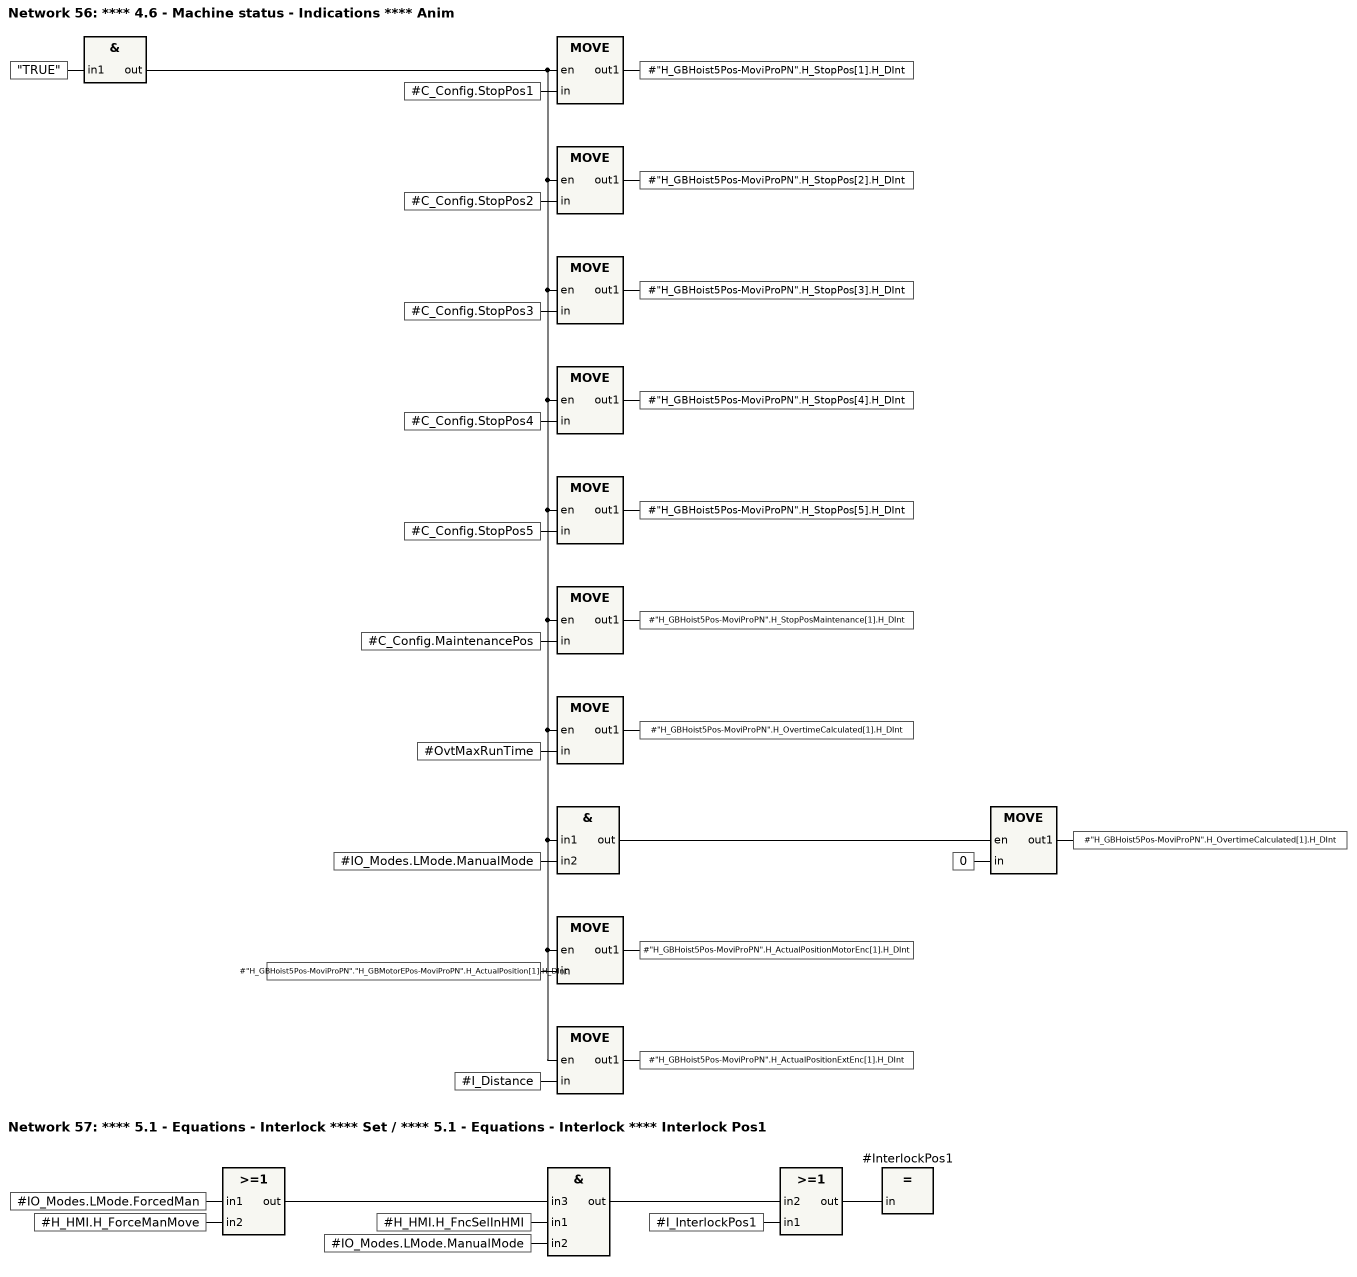
   IF "TRUE" THEN
       #"H_GBHoist5Pos-MoviProPN".H_StopPos[1].H_DInt := #C_Config.StopPos1;
       #"H_GBHoist5Pos-MoviProPN".H_StopPos[2].H_DInt := #C_Config.StopPos2;
       #"H_GBHoist5Pos-MoviProPN".H_StopPos[3].H_DInt := #C_Config.StopPos3;
       #"H_GBHoist5Pos-MoviProPN".H_StopPos[4].H_DInt := #C_Config.StopPos4;
       #"H_GBHoist5Pos-MoviProPN".H_StopPos[5].H_DInt := #C_Config.StopPos5;
       #"H_GBHoist5Pos-MoviProPN".H_StopPosMaintenance[1].H_DInt := #C_Config.MaintenancePos;
       #"H_GBHoist5Pos-MoviProPN".H_OvertimeCalculated[1].H_DInt := #OvtMaxRunTime;
   END_IF;
   IF "TRUE" AND #IO_Modes.LMode.ManualMode THEN
       #"H_GBHoist5Pos-MoviProPN".H_OvertimeCalculated[1].H_DInt := 0;
   END_IF;
   IF "TRUE" THEN
       #"H_GBHoist5Pos-MoviProPN".H_ActualPositionMotorEnc[1].H_DInt := #"H_GBHoist5Pos-MoviProPN"."H_GBMotorEPos-MoviProPN".H_ActualPosition[1].H_DInt;
       #"H_GBHoist5Pos-MoviProPN".H_ActualPositionExtEnc[1].H_DInt := #I_Distance;
   END_IF;
END_REGION

REGION Network 57: **** 5.1 - Equations - Interlock **** Set / **** 5.1 - Equations - Interlock **** Interlock Pos1
   // Interlock
   #InterlockPos1 := ((#IO_Modes.LMode.ForcedMan OR #H_HMI.H_ForceManMove) AND #H_HMI.H_FncSelInHMI AND #IO_Modes.LMode.ManualMode) OR #I_InterlockPos1;
END_REGION

REGION Network 58: **** 5.1 - Equations - Interlock **** Set / **** 5.1 - Equations - Interlock **** Interlock Pos2
   // Interlock
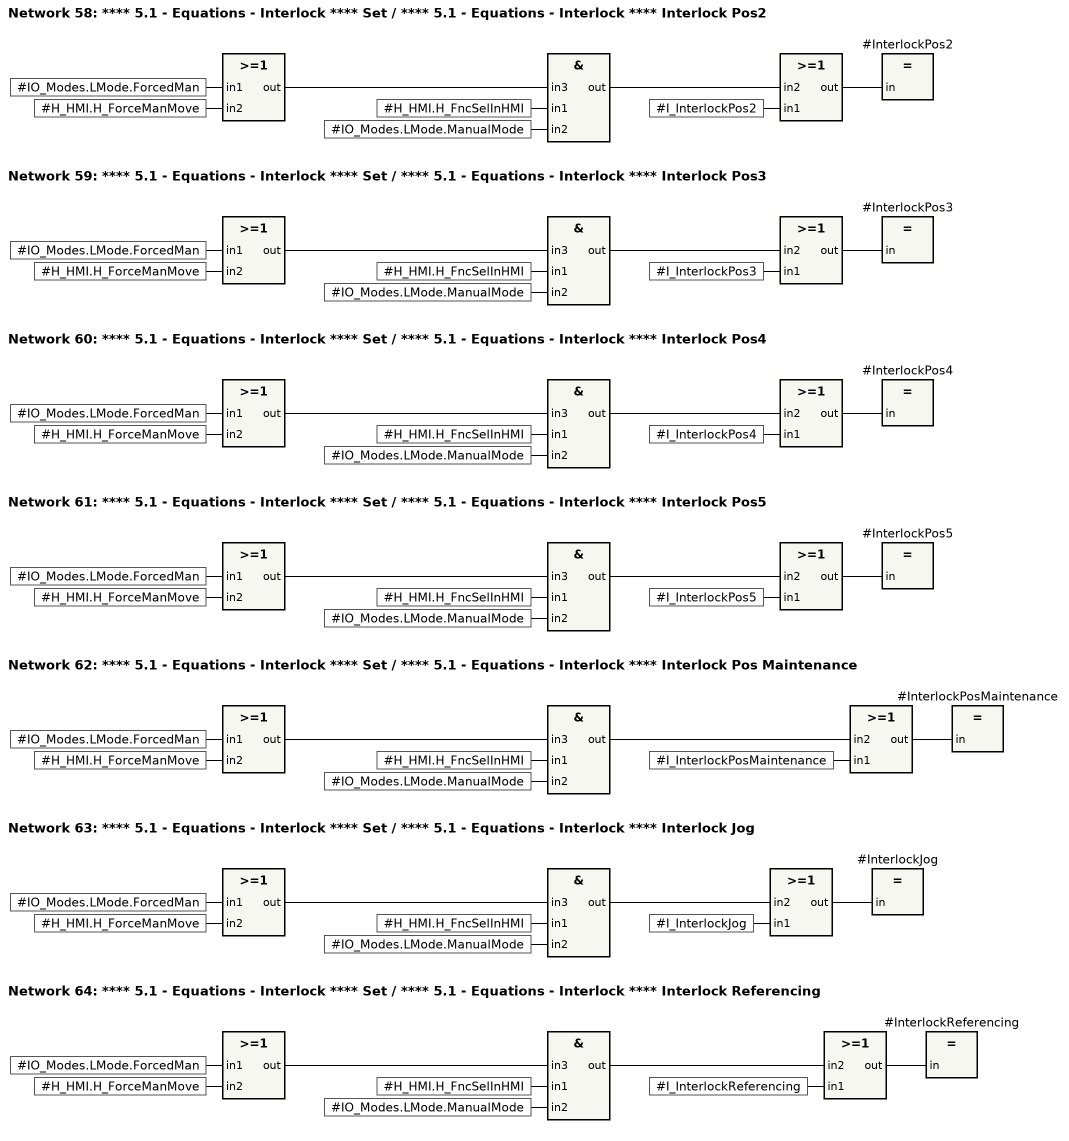
   #InterlockPos2 := ((#IO_Modes.LMode.ForcedMan OR #H_HMI.H_ForceManMove) AND #H_HMI.H_FncSelInHMI AND #IO_Modes.LMode.ManualMode) OR #I_InterlockPos2;
END_REGION

REGION Network 59: **** 5.1 - Equations - Interlock **** Set / **** 5.1 - Equations - Interlock **** Interlock Pos3
   // Interlock
   #InterlockPos3 := ((#IO_Modes.LMode.ForcedMan OR #H_HMI.H_ForceManMove) AND #H_HMI.H_FncSelInHMI AND #IO_Modes.LMode.ManualMode) OR #I_InterlockPos3;
END_REGION

REGION Network 60: **** 5.1 - Equations - Interlock **** Set / **** 5.1 - Equations - Interlock **** Interlock Pos4
   // Interlock
   #InterlockPos4 := ((#IO_Modes.LMode.ForcedMan OR #H_HMI.H_ForceManMove) AND #H_HMI.H_FncSelInHMI AND #IO_Modes.LMode.ManualMode) OR #I_InterlockPos4;
END_REGION

REGION Network 61: **** 5.1 - Equations - Interlock **** Set / **** 5.1 - Equations - Interlock **** Interlock Pos5
   // Interlock
   #InterlockPos5 := ((#IO_Modes.LMode.ForcedMan OR #H_HMI.H_ForceManMove) AND #H_HMI.H_FncSelInHMI AND #IO_Modes.LMode.ManualMode) OR #I_InterlockPos5;
END_REGION

REGION Network 62: **** 5.1 - Equations - Interlock **** Set / **** 5.1 - Equations - Interlock **** Interlock Pos Maintenance
   // Interlock
   #InterlockPosMaintenance := ((#IO_Modes.LMode.ForcedMan OR #H_HMI.H_ForceManMove) AND #H_HMI.H_FncSelInHMI AND #IO_Modes.LMode.ManualMode) OR #I_InterlockPosMaintenance;
END_REGION

REGION Network 63: **** 5.1 - Equations - Interlock **** Set / **** 5.1 - Equations - Interlock **** Interlock Jog
   // Interlock
   #InterlockJog := ((#IO_Modes.LMode.ForcedMan OR #H_HMI.H_ForceManMove) AND #H_HMI.H_FncSelInHMI AND #IO_Modes.LMode.ManualMode) OR #I_InterlockJog;
END_REGION

REGION Network 64: **** 5.1 - Equations - Interlock **** Set / **** 5.1 - Equations - Interlock **** Interlock Referencing
   // Interlock
   #InterlockReferencing := ((#IO_Modes.LMode.ForcedMan OR #H_HMI.H_ForceManMove) AND #H_HMI.H_FncSelInHMI AND #IO_Modes.LMode.ManualMode) OR #I_InterlockReferencing;
END_REGION

REGION Network 65: **** 5.2 - Equations - Equations **** Epos Cmd
   // Drive is steered by EPos commands
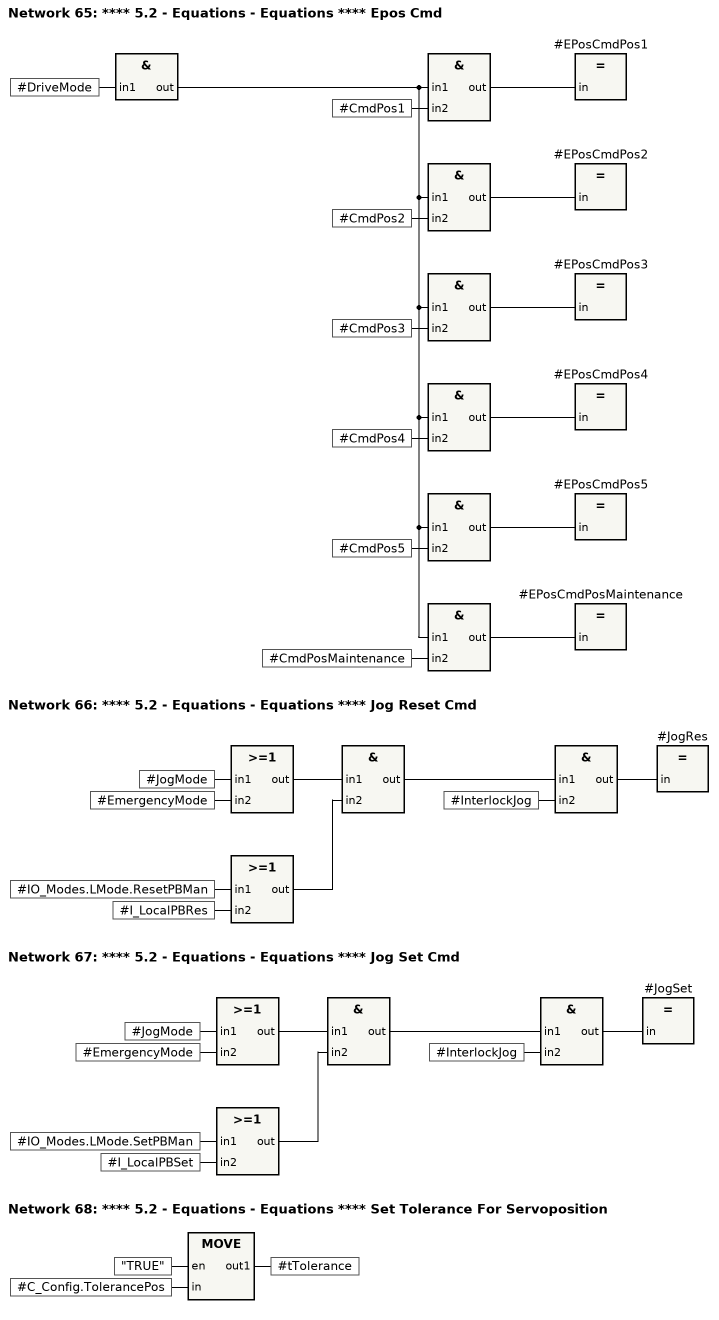
   #EPosCmdPos1 := #DriveMode AND #CmdPos1;
   #EPosCmdPos2 := #DriveMode AND #CmdPos2;
   #EPosCmdPos3 := #DriveMode AND #CmdPos3;
   #EPosCmdPos4 := #DriveMode AND #CmdPos4;
   #EPosCmdPos5 := #DriveMode AND #CmdPos5;
   #EPosCmdPosMaintenance := #DriveMode AND #CmdPosMaintenance;
END_REGION

REGION Network 66: **** 5.2 - Equations - Equations **** Jog Reset Cmd
   // Drive is steered by Jog commands in reset direction
   #JogRes := (#JogMode OR #EmergencyMode) AND (#IO_Modes.LMode.ResetPBMan OR #I_LocalPBRes) AND #InterlockJog;
END_REGION

REGION Network 67: **** 5.2 - Equations - Equations **** Jog Set Cmd
   // Drive is steered by Jog commands in set direction
   #JogSet := (#JogMode OR #EmergencyMode) AND (#IO_Modes.LMode.SetPBMan OR #I_LocalPBSet) AND #InterlockJog;
END_REGION

REGION Network 68: **** 5.2 - Equations - Equations **** Set Tolerance For Servoposition
   // Set Tolerance For ServoPosition
   IF "TRUE" THEN #tTolerance := #C_Config.TolerancePos; END_IF;
END_REGION

REGION Network 69: **** 5.2 - Equations - Equations **** Calculate Tolerance Index Pos 1
   // Calculate Tolerance Index Pos 1
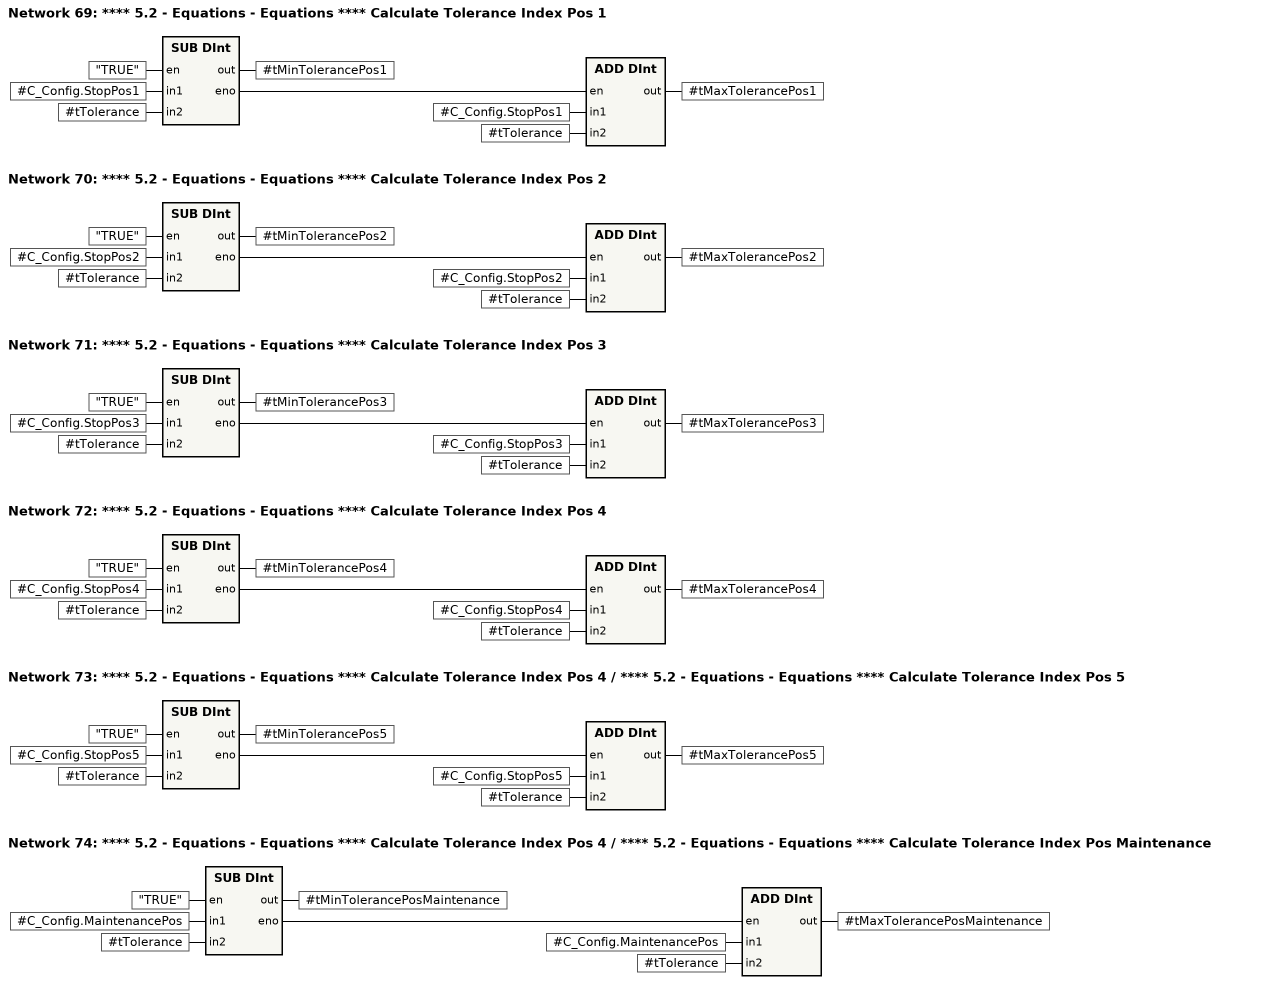
   // ENO of a box is taken as its EN; it also drops when the box reports an error
   IF "TRUE" THEN
       #tMinTolerancePos1 := #C_Config.StopPos1 - #tTolerance;
       #tMaxTolerancePos1 := #C_Config.StopPos1 + #tTolerance;
   END_IF;
END_REGION

REGION Network 70: **** 5.2 - Equations - Equations **** Calculate Tolerance Index Pos 2
   // Calculate Tolerance Index Pos 2
   // ENO of a box is taken as its EN; it also drops when the box reports an error
   IF "TRUE" THEN
       #tMinTolerancePos2 := #C_Config.StopPos2 - #tTolerance;
       #tMaxTolerancePos2 := #C_Config.StopPos2 + #tTolerance;
   END_IF;
END_REGION

REGION Network 71: **** 5.2 - Equations - Equations **** Calculate Tolerance Index Pos 3
   // Calculate Tolerance Index Pos 3
   // ENO of a box is taken as its EN; it also drops when the box reports an error
   IF "TRUE" THEN
       #tMinTolerancePos3 := #C_Config.StopPos3 - #tTolerance;
       #tMaxTolerancePos3 := #C_Config.StopPos3 + #tTolerance;
   END_IF;
END_REGION

REGION Network 72: **** 5.2 - Equations - Equations **** Calculate Tolerance Index Pos 4
   // Calculate Tolerance Index Pos 4
   // ENO of a box is taken as its EN; it also drops when the box reports an error
   IF "TRUE" THEN
       #tMinTolerancePos4 := #C_Config.StopPos4 - #tTolerance;
       #tMaxTolerancePos4 := #C_Config.StopPos4 + #tTolerance;
   END_IF;
END_REGION

REGION Network 73: **** 5.2 - Equations - Equations **** Calculate Tolerance Index Pos 4 / **** 5.2 - Equations - Equations **** Calculate Tolerance Index Pos 5
   // Calculate Tolerance Index Pos 4 / Calculate Tolerance Index Pos 5
   // ENO of a box is taken as its EN; it also drops when the box reports an error
   IF "TRUE" THEN
       #tMinTolerancePos5 := #C_Config.StopPos5 - #tTolerance;
       #tMaxTolerancePos5 := #C_Config.StopPos5 + #tTolerance;
   END_IF;
END_REGION

REGION Network 74: **** 5.2 - Equations - Equations **** Calculate Tolerance Index Pos 4 / **** 5.2 - Equations - Equations **** Calculate Tolerance Index Pos Maintenance
   // Calculate Tolerance Index Pos 4 / Calculate Tolerance Index Pos Maintenance
   // ENO of a box is taken as its EN; it also drops when the box reports an error
   IF "TRUE" THEN
       #tMinTolerancePosMaintenance := #C_Config.MaintenancePos - #tTolerance;
       #tMaxTolerancePosMaintenance := #C_Config.MaintenancePos + #tTolerance;
   END_IF;
END_REGION

REGION Network 75: **** 5.2 - Equations - Equations **** Alarm Condition Keep Position 1
   // Alarm Condition Keep Position
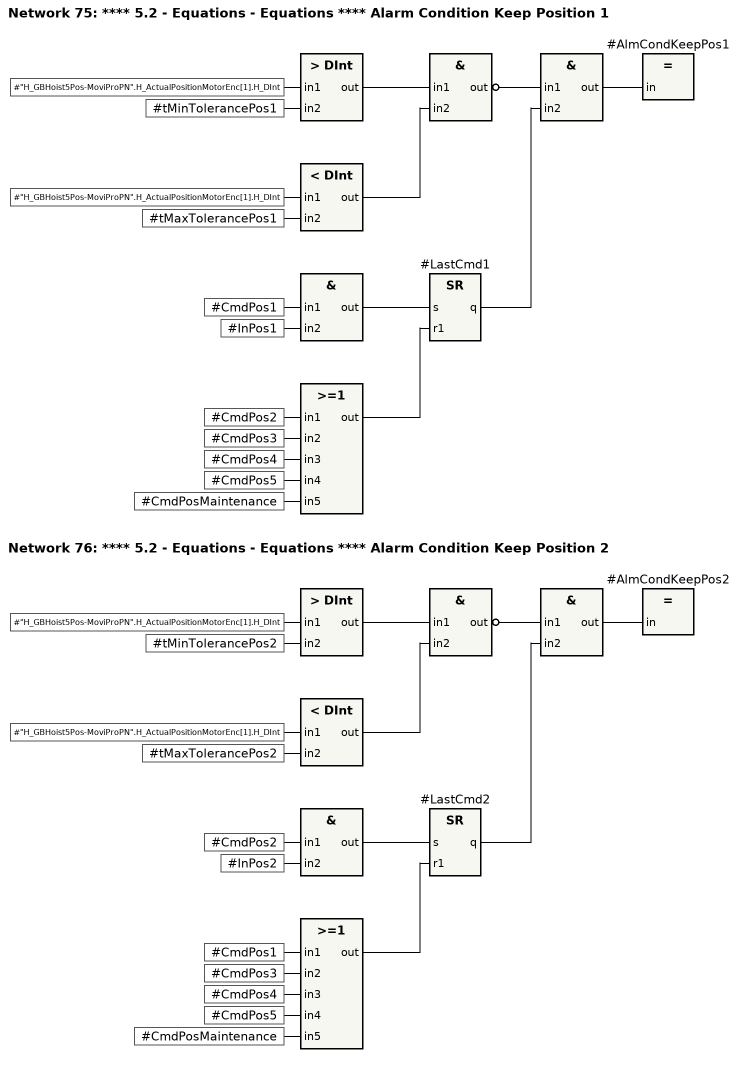
   IF #CmdPos1 AND #InPos1 THEN
       #LastCmd1 := TRUE;   // SR flip-flop
   END_IF;
   IF #CmdPos2 OR #CmdPos3 OR #CmdPos4 OR #CmdPos5 OR #CmdPosMaintenance THEN #LastCmd1 := FALSE; END_IF;
   #AlmCondKeepPos1 := NOT ((#"H_GBHoist5Pos-MoviProPN".H_ActualPositionMotorEnc[1].H_DInt > #tMinTolerancePos1) AND (#"H_GBHoist5Pos-MoviProPN".H_ActualPositionMotorEnc[1].H_DInt < #tMaxTolerancePos1)) AND #LastCmd1;
END_REGION

REGION Network 76: **** 5.2 - Equations - Equations **** Alarm Condition Keep Position 2
   // Alarm Condition Keep Position
   IF #CmdPos2 AND #InPos2 THEN
       #LastCmd2 := TRUE;   // SR flip-flop
   END_IF;
   IF #CmdPos1 OR #CmdPos3 OR #CmdPos4 OR #CmdPos5 OR #CmdPosMaintenance THEN #LastCmd2 := FALSE; END_IF;
   #AlmCondKeepPos2 := NOT ((#"H_GBHoist5Pos-MoviProPN".H_ActualPositionMotorEnc[1].H_DInt > #tMinTolerancePos2) AND (#"H_GBHoist5Pos-MoviProPN".H_ActualPositionMotorEnc[1].H_DInt < #tMaxTolerancePos2)) AND #LastCmd2;
END_REGION

REGION Network 77: **** 5.2 - Equations - Equations **** Alarm Condition Keep Position 3
   // Alarm Condition Keep Position
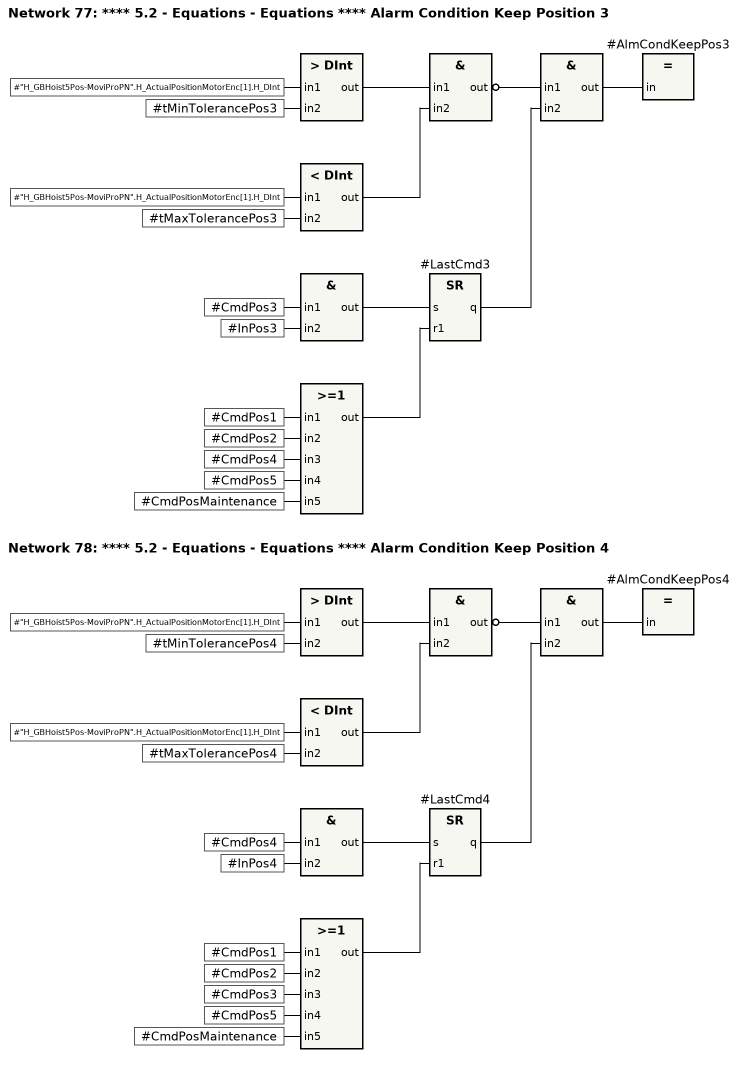
   IF #CmdPos3 AND #InPos3 THEN
       #LastCmd3 := TRUE;   // SR flip-flop
   END_IF;
   IF #CmdPos1 OR #CmdPos2 OR #CmdPos4 OR #CmdPos5 OR #CmdPosMaintenance THEN #LastCmd3 := FALSE; END_IF;
   #AlmCondKeepPos3 := NOT ((#"H_GBHoist5Pos-MoviProPN".H_ActualPositionMotorEnc[1].H_DInt > #tMinTolerancePos3) AND (#"H_GBHoist5Pos-MoviProPN".H_ActualPositionMotorEnc[1].H_DInt < #tMaxTolerancePos3)) AND #LastCmd3;
END_REGION

REGION Network 78: **** 5.2 - Equations - Equations **** Alarm Condition Keep Position 4
   // Alarm Condition Keep Position
   IF #CmdPos4 AND #InPos4 THEN
       #LastCmd4 := TRUE;   // SR flip-flop
   END_IF;
   IF #CmdPos1 OR #CmdPos2 OR #CmdPos3 OR #CmdPos5 OR #CmdPosMaintenance THEN #LastCmd4 := FALSE; END_IF;
   #AlmCondKeepPos4 := NOT ((#"H_GBHoist5Pos-MoviProPN".H_ActualPositionMotorEnc[1].H_DInt > #tMinTolerancePos4) AND (#"H_GBHoist5Pos-MoviProPN".H_ActualPositionMotorEnc[1].H_DInt < #tMaxTolerancePos4)) AND #LastCmd4;
END_REGION

REGION Network 79: **** 5.2 - Equations - Equations **** Alarm Condition Keep Position 4 / **** 5.2 - Equations - Equations **** Alarm Condition Keep Position 5
   // Alarm Condition Keep Position
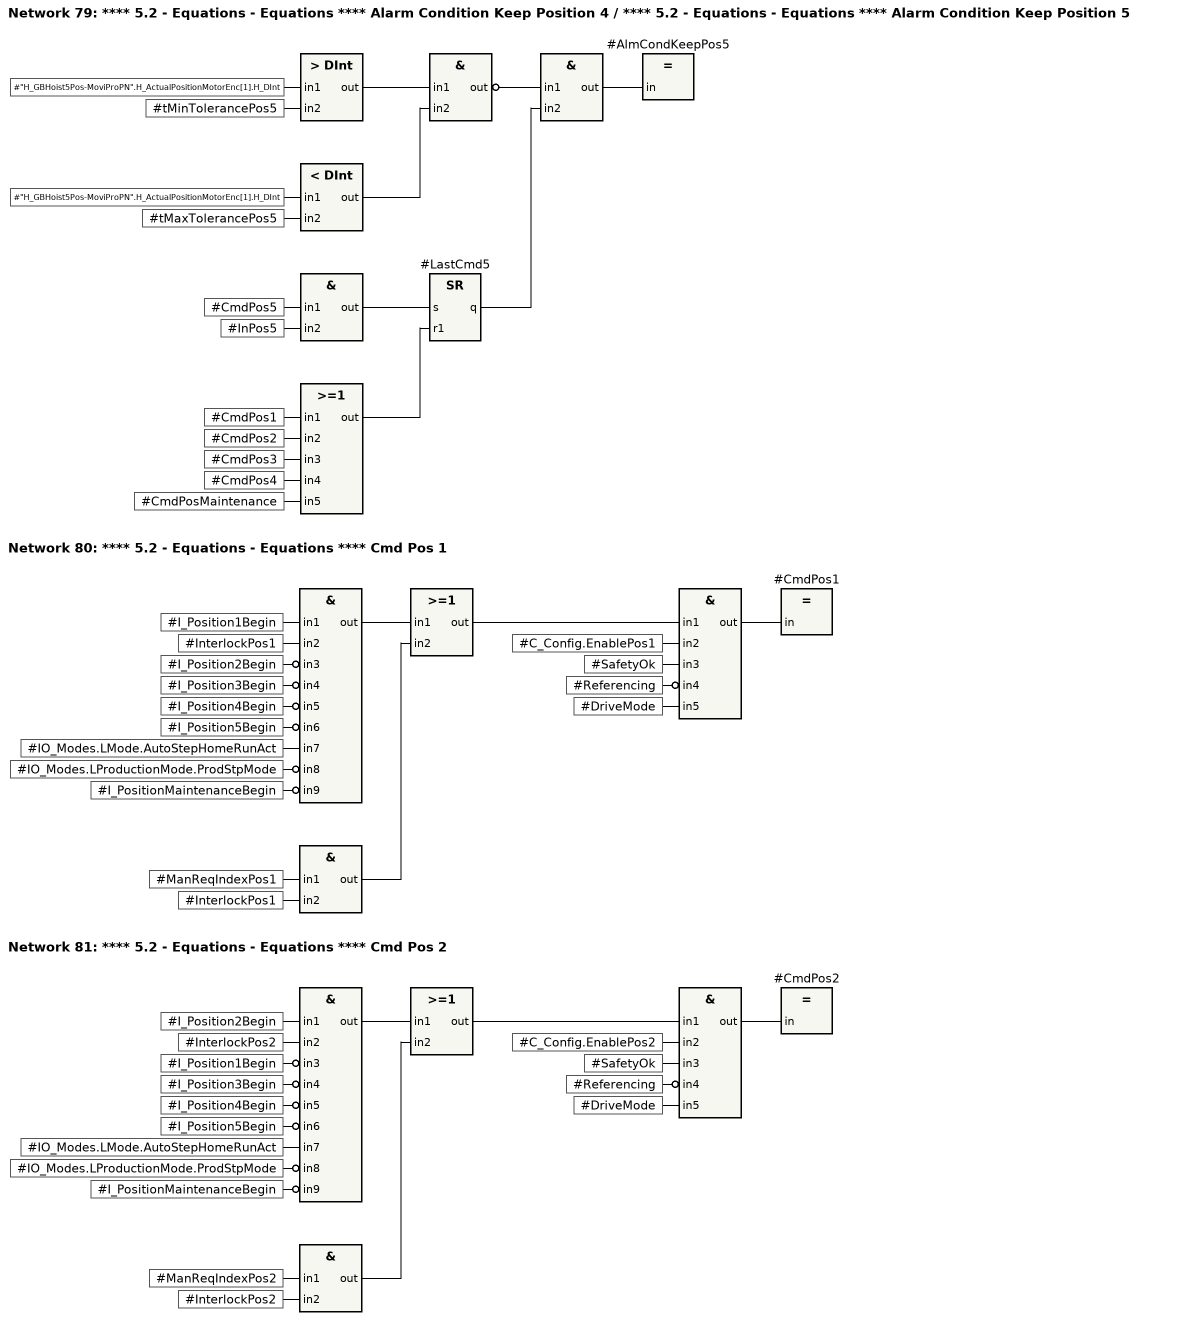
   IF #CmdPos5 AND #InPos5 THEN
       #LastCmd5 := TRUE;   // SR flip-flop
   END_IF;
   IF #CmdPos1 OR #CmdPos2 OR #CmdPos3 OR #CmdPos4 OR #CmdPosMaintenance THEN #LastCmd5 := FALSE; END_IF;
   #AlmCondKeepPos5 := NOT ((#"H_GBHoist5Pos-MoviProPN".H_ActualPositionMotorEnc[1].H_DInt > #tMinTolerancePos5) AND (#"H_GBHoist5Pos-MoviProPN".H_ActualPositionMotorEnc[1].H_DInt < #tMaxTolerancePos5)) AND #LastCmd5;
END_REGION

REGION Network 80: **** 5.2 - Equations - Equations **** Cmd Pos 1
   // Cmd Pos 1
   #CmdPos1 := ((#I_Position1Begin AND #InterlockPos1 AND NOT #I_Position2Begin AND NOT #I_Position3Begin AND NOT #I_Position4Begin AND NOT #I_Position5Begin AND #IO_Modes.LMode.AutoStepHomeRunAct AND NOT #IO_Modes.LProductionMode.ProdStpMode AND NOT #I_PositionMaintenanceBegin) OR (#ManReqIndexPos1 AND #InterlockPos1)) AND #C_Config.EnablePos1 AND #SafetyOk AND NOT #Referencing AND #DriveMode;
END_REGION

REGION Network 81: **** 5.2 - Equations - Equations **** Cmd Pos 2
   // Cmd Pos 2
   #CmdPos2 := ((#I_Position2Begin AND #InterlockPos2 AND NOT #I_Position1Begin AND NOT #I_Position3Begin AND NOT #I_Position4Begin AND NOT #I_Position5Begin AND #IO_Modes.LMode.AutoStepHomeRunAct AND NOT #IO_Modes.LProductionMode.ProdStpMode AND NOT #I_PositionMaintenanceBegin) OR (#ManReqIndexPos2 AND #InterlockPos2)) AND #C_Config.EnablePos2 AND #SafetyOk AND NOT #Referencing AND #DriveMode;
END_REGION

REGION Network 82: **** 5.2 - Equations - Equations **** Cmd Pos 3
   // Cmd Pos 3
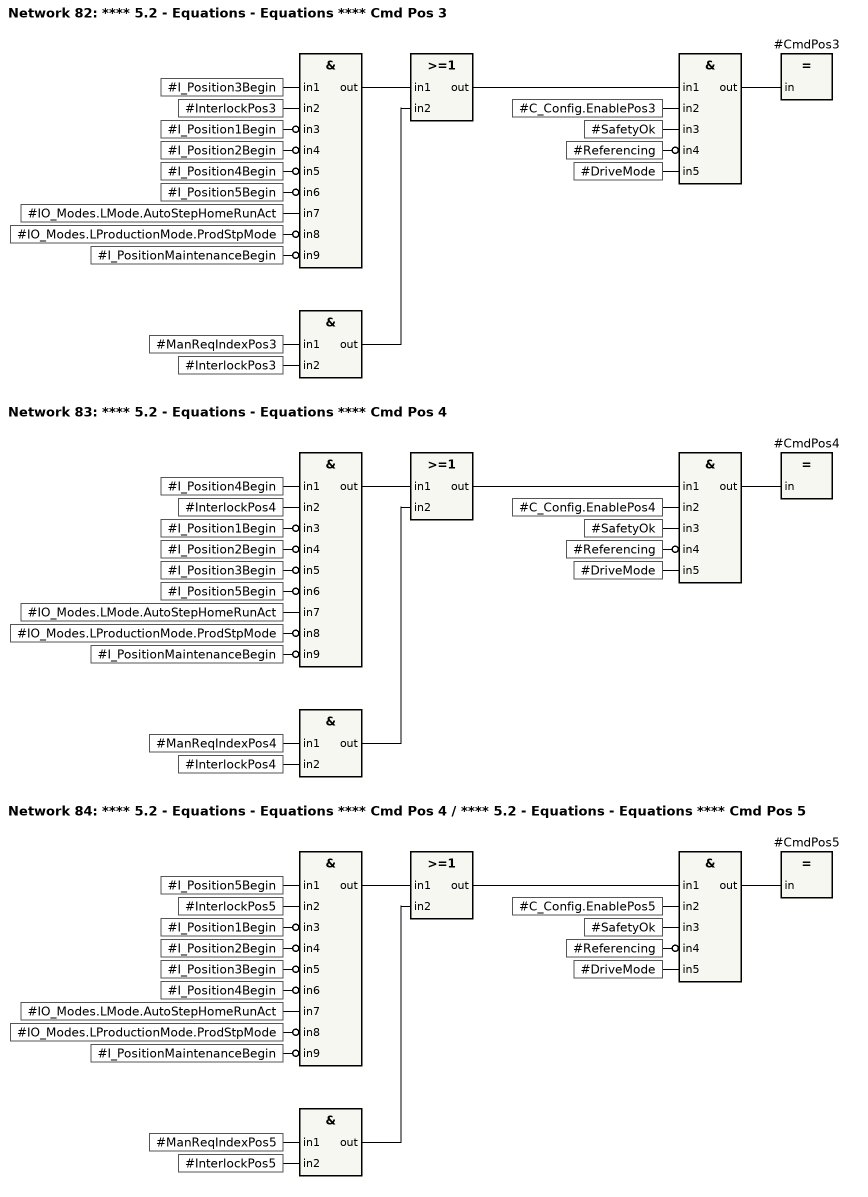
   #CmdPos3 := ((#I_Position3Begin AND #InterlockPos3 AND NOT #I_Position1Begin AND NOT #I_Position2Begin AND NOT #I_Position4Begin AND NOT #I_Position5Begin AND #IO_Modes.LMode.AutoStepHomeRunAct AND NOT #IO_Modes.LProductionMode.ProdStpMode AND NOT #I_PositionMaintenanceBegin) OR (#ManReqIndexPos3 AND #InterlockPos3)) AND #C_Config.EnablePos3 AND #SafetyOk AND NOT #Referencing AND #DriveMode;
END_REGION

REGION Network 83: **** 5.2 - Equations - Equations **** Cmd Pos 4
   // Cmd Pos 4
   #CmdPos4 := ((#I_Position4Begin AND #InterlockPos4 AND NOT #I_Position1Begin AND NOT #I_Position2Begin AND NOT #I_Position3Begin AND NOT #I_Position5Begin AND #IO_Modes.LMode.AutoStepHomeRunAct AND NOT #IO_Modes.LProductionMode.ProdStpMode AND NOT #I_PositionMaintenanceBegin) OR (#ManReqIndexPos4 AND #InterlockPos4)) AND #C_Config.EnablePos4 AND #SafetyOk AND NOT #Referencing AND #DriveMode;
END_REGION

REGION Network 84: **** 5.2 - Equations - Equations **** Cmd Pos 4 / **** 5.2 - Equations - Equations **** Cmd Pos 5
   // Cmd Pos 4
   #CmdPos5 := ((#I_Position5Begin AND #InterlockPos5 AND NOT #I_Position1Begin AND NOT #I_Position2Begin AND NOT #I_Position3Begin AND NOT #I_Position4Begin AND #IO_Modes.LMode.AutoStepHomeRunAct AND NOT #IO_Modes.LProductionMode.ProdStpMode AND NOT #I_PositionMaintenanceBegin) OR (#ManReqIndexPos5 AND #InterlockPos5)) AND #C_Config.EnablePos5 AND #SafetyOk AND NOT #Referencing AND #DriveMode;
END_REGION

REGION Network 85: **** 5.2 - Equations - Equations **** Cmd Pos 4 / **** 5.2 - Equations - Equations **** Cmd Pos Maintenance
   // Cmd Pos 4 / Cmd Pos Maintenance
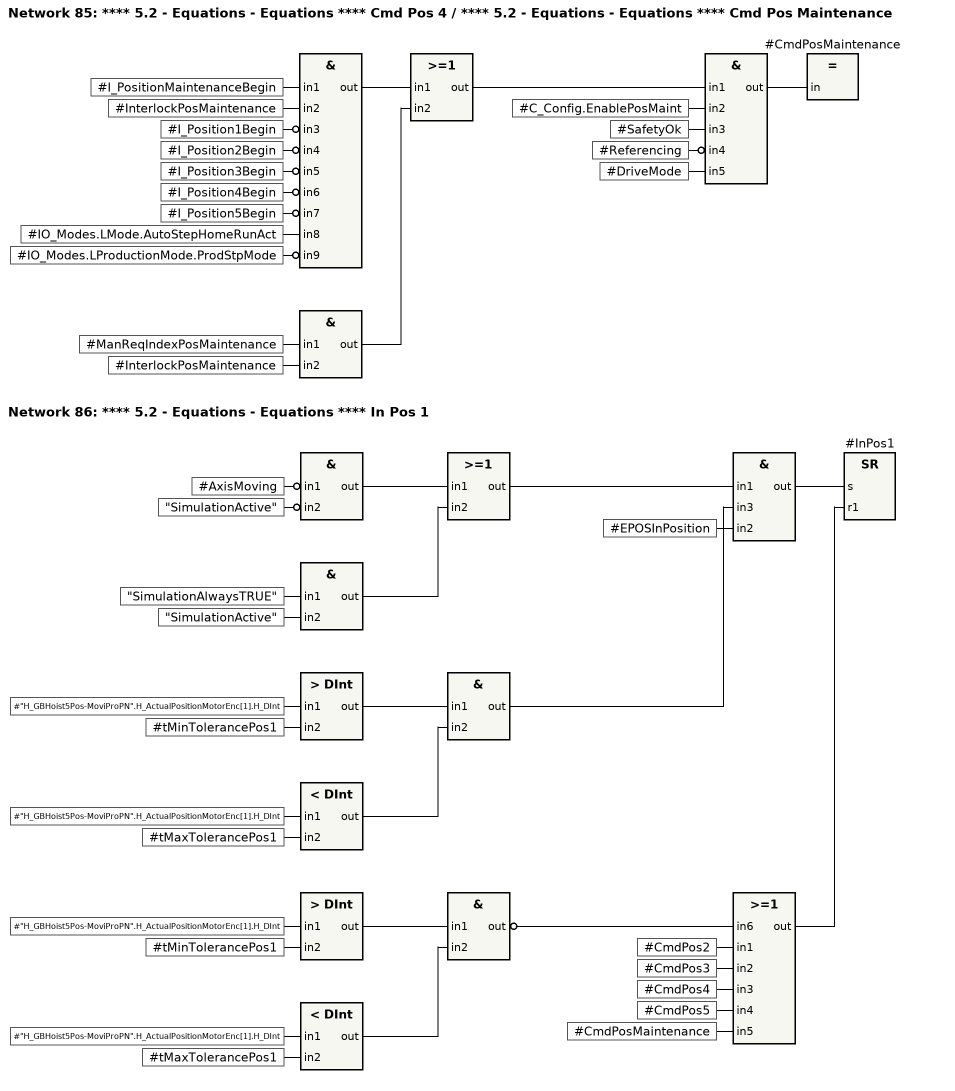
   #CmdPosMaintenance := ((#I_PositionMaintenanceBegin AND #InterlockPosMaintenance AND NOT #I_Position1Begin AND NOT #I_Position2Begin AND NOT #I_Position3Begin AND NOT #I_Position4Begin AND NOT #I_Position5Begin AND #IO_Modes.LMode.AutoStepHomeRunAct AND NOT #IO_Modes.LProductionMode.ProdStpMode) OR (#ManReqIndexPosMaintenance AND #InterlockPosMaintenance)) AND #C_Config.EnablePosMaint AND #SafetyOk AND NOT #Referencing AND #DriveMode;
END_REGION

REGION Network 86: **** 5.2 - Equations - Equations **** In Pos 1
   // In Pos 1
   IF ((NOT #AxisMoving AND NOT "SimulationActive") OR ("SimulationAlwaysTRUE" AND "SimulationActive")) AND (#"H_GBHoist5Pos-MoviProPN".H_ActualPositionMotorEnc[1].H_DInt > #tMinTolerancePos1) AND (#"H_GBHoist5Pos-MoviProPN".H_ActualPositionMotorEnc[1].H_DInt < #tMaxTolerancePos1) AND #EPOSInPosition THEN
       #InPos1 := TRUE;   // SR flip-flop
   END_IF;
   IF NOT ((#"H_GBHoist5Pos-MoviProPN".H_ActualPositionMotorEnc[1].H_DInt > #tMinTolerancePos1) AND (#"H_GBHoist5Pos-MoviProPN".H_ActualPositionMotorEnc[1].H_DInt < #tMaxTolerancePos1)) OR #CmdPos2 OR #CmdPos3 OR #CmdPos4 OR #CmdPos5 OR #CmdPosMaintenance THEN
       #InPos1 := FALSE;
   END_IF;
END_REGION

REGION Network 87: **** 5.2 - Equations - Equations **** In Pos 2
   // In Pos 2
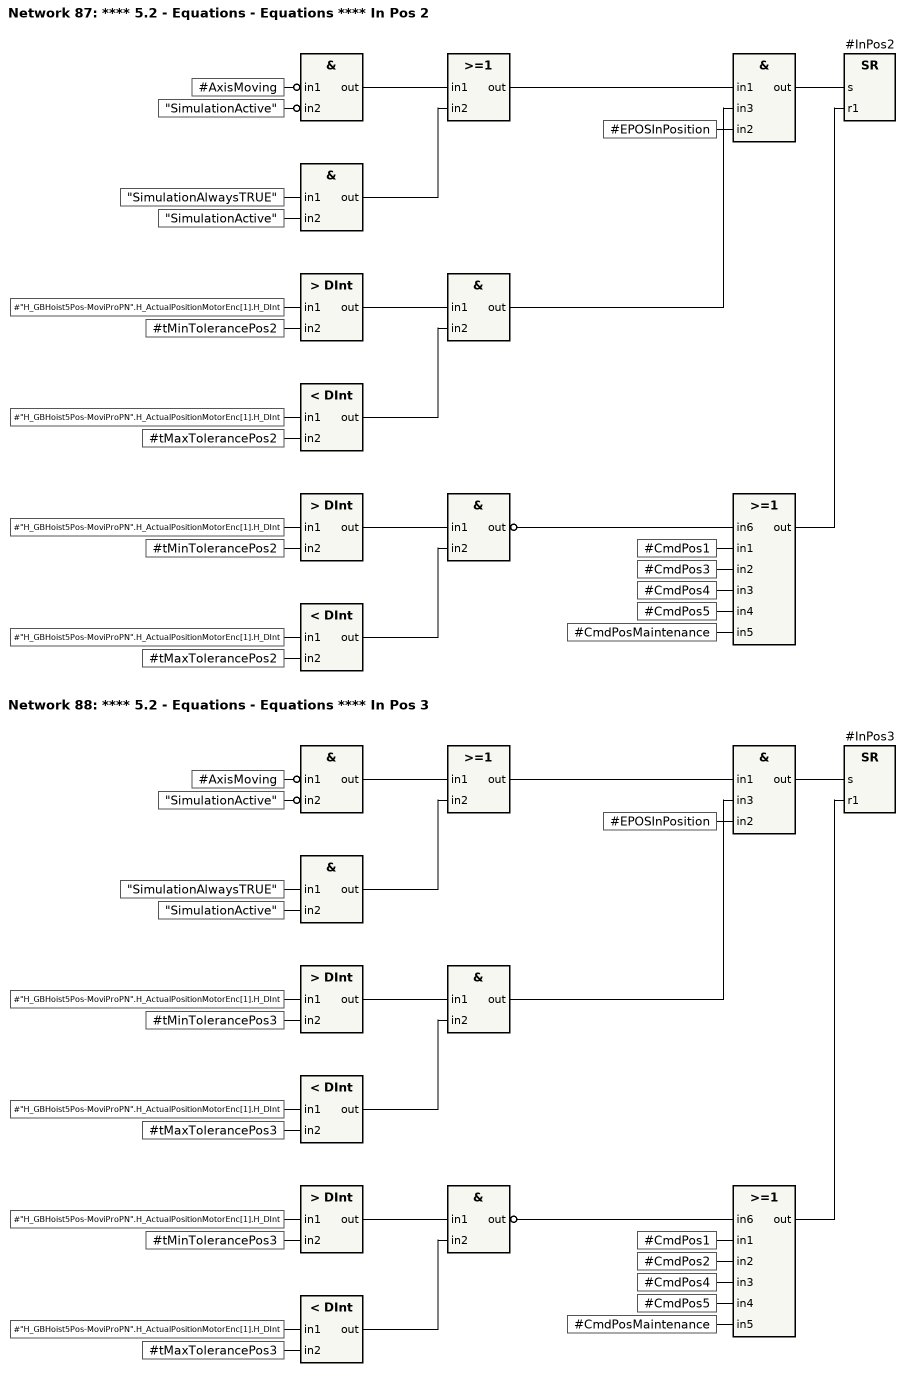
   IF ((NOT #AxisMoving AND NOT "SimulationActive") OR ("SimulationAlwaysTRUE" AND "SimulationActive")) AND (#"H_GBHoist5Pos-MoviProPN".H_ActualPositionMotorEnc[1].H_DInt > #tMinTolerancePos2) AND (#"H_GBHoist5Pos-MoviProPN".H_ActualPositionMotorEnc[1].H_DInt < #tMaxTolerancePos2) AND #EPOSInPosition THEN
       #InPos2 := TRUE;   // SR flip-flop
   END_IF;
   IF NOT ((#"H_GBHoist5Pos-MoviProPN".H_ActualPositionMotorEnc[1].H_DInt > #tMinTolerancePos2) AND (#"H_GBHoist5Pos-MoviProPN".H_ActualPositionMotorEnc[1].H_DInt < #tMaxTolerancePos2)) OR #CmdPos1 OR #CmdPos3 OR #CmdPos4 OR #CmdPos5 OR #CmdPosMaintenance THEN
       #InPos2 := FALSE;
   END_IF;
END_REGION

REGION Network 88: **** 5.2 - Equations - Equations **** In Pos 3
   // In Pos 3
   IF ((NOT #AxisMoving AND NOT "SimulationActive") OR ("SimulationAlwaysTRUE" AND "SimulationActive")) AND (#"H_GBHoist5Pos-MoviProPN".H_ActualPositionMotorEnc[1].H_DInt > #tMinTolerancePos3) AND (#"H_GBHoist5Pos-MoviProPN".H_ActualPositionMotorEnc[1].H_DInt < #tMaxTolerancePos3) AND #EPOSInPosition THEN
       #InPos3 := TRUE;   // SR flip-flop
   END_IF;
   IF NOT ((#"H_GBHoist5Pos-MoviProPN".H_ActualPositionMotorEnc[1].H_DInt > #tMinTolerancePos3) AND (#"H_GBHoist5Pos-MoviProPN".H_ActualPositionMotorEnc[1].H_DInt < #tMaxTolerancePos3)) OR #CmdPos1 OR #CmdPos2 OR #CmdPos4 OR #CmdPos5 OR #CmdPosMaintenance THEN
       #InPos3 := FALSE;
   END_IF;
END_REGION

REGION Network 89: **** 5.2 - Equations - Equations **** In Pos 4
   // In Pos 4
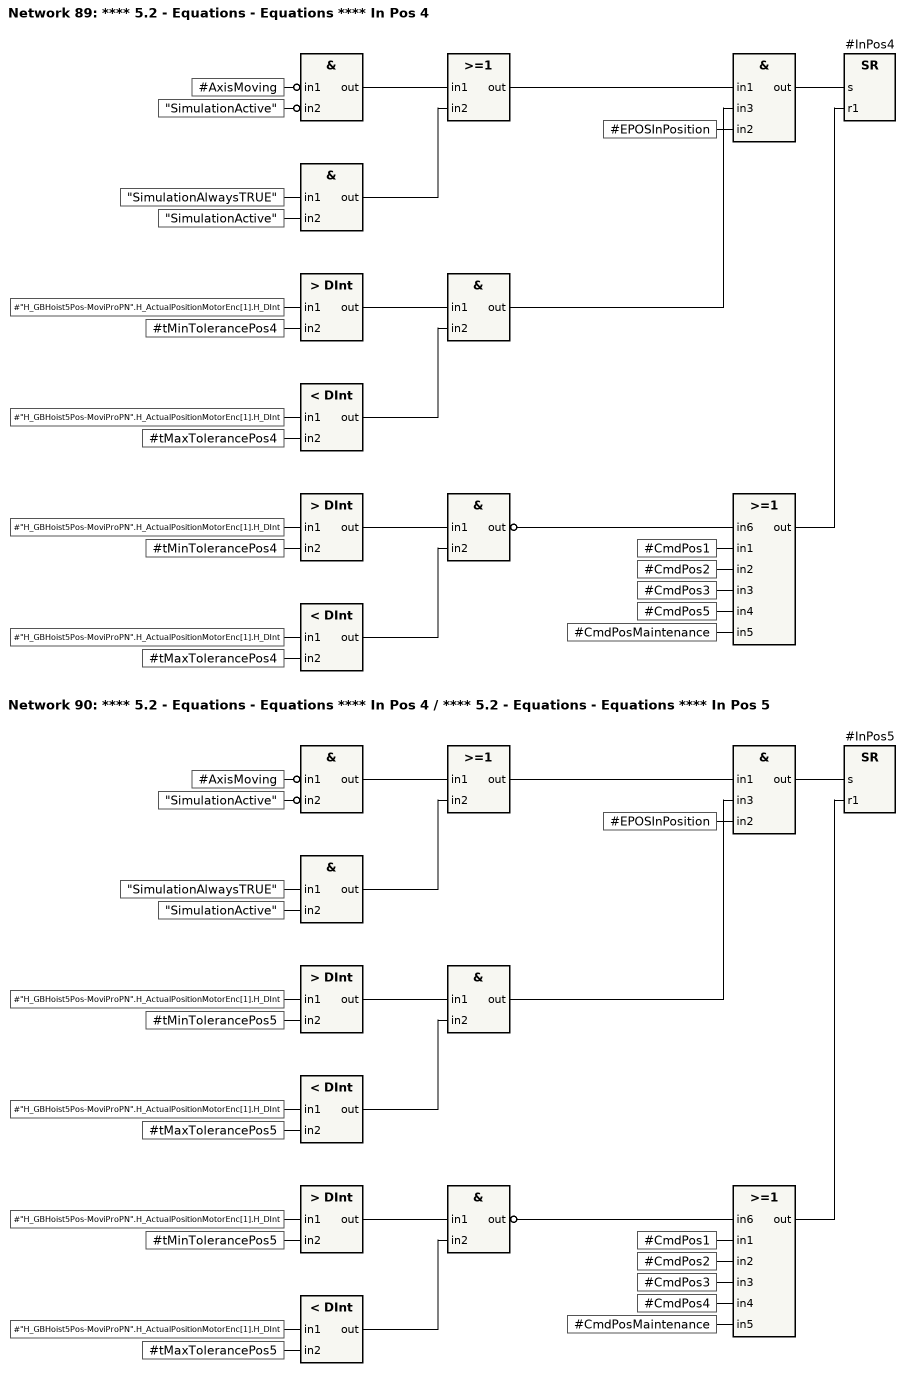
   IF ((NOT #AxisMoving AND NOT "SimulationActive") OR ("SimulationAlwaysTRUE" AND "SimulationActive")) AND (#"H_GBHoist5Pos-MoviProPN".H_ActualPositionMotorEnc[1].H_DInt > #tMinTolerancePos4) AND (#"H_GBHoist5Pos-MoviProPN".H_ActualPositionMotorEnc[1].H_DInt < #tMaxTolerancePos4) AND #EPOSInPosition THEN
       #InPos4 := TRUE;   // SR flip-flop
   END_IF;
   IF NOT ((#"H_GBHoist5Pos-MoviProPN".H_ActualPositionMotorEnc[1].H_DInt > #tMinTolerancePos4) AND (#"H_GBHoist5Pos-MoviProPN".H_ActualPositionMotorEnc[1].H_DInt < #tMaxTolerancePos4)) OR #CmdPos1 OR #CmdPos2 OR #CmdPos3 OR #CmdPos5 OR #CmdPosMaintenance THEN
       #InPos4 := FALSE;
   END_IF;
END_REGION

REGION Network 90: **** 5.2 - Equations - Equations **** In Pos 4 / **** 5.2 - Equations - Equations **** In Pos 5
   // In Pos 4 / In Pos 5
   IF ((NOT #AxisMoving AND NOT "SimulationActive") OR ("SimulationAlwaysTRUE" AND "SimulationActive")) AND (#"H_GBHoist5Pos-MoviProPN".H_ActualPositionMotorEnc[1].H_DInt > #tMinTolerancePos5) AND (#"H_GBHoist5Pos-MoviProPN".H_ActualPositionMotorEnc[1].H_DInt < #tMaxTolerancePos5) AND #EPOSInPosition THEN
       #InPos5 := TRUE;   // SR flip-flop
   END_IF;
   IF NOT ((#"H_GBHoist5Pos-MoviProPN".H_ActualPositionMotorEnc[1].H_DInt > #tMinTolerancePos5) AND (#"H_GBHoist5Pos-MoviProPN".H_ActualPositionMotorEnc[1].H_DInt < #tMaxTolerancePos5)) OR #CmdPos1 OR #CmdPos2 OR #CmdPos3 OR #CmdPos4 OR #CmdPosMaintenance THEN
       #InPos5 := FALSE;
   END_IF;
END_REGION

REGION Network 91: **** 5.2 - Equations - Equations **** In Pos 4 / **** 5.2 - Equations - Equations **** In Pos Maintenance
   // In Pos 4 / In Pos Maintenance
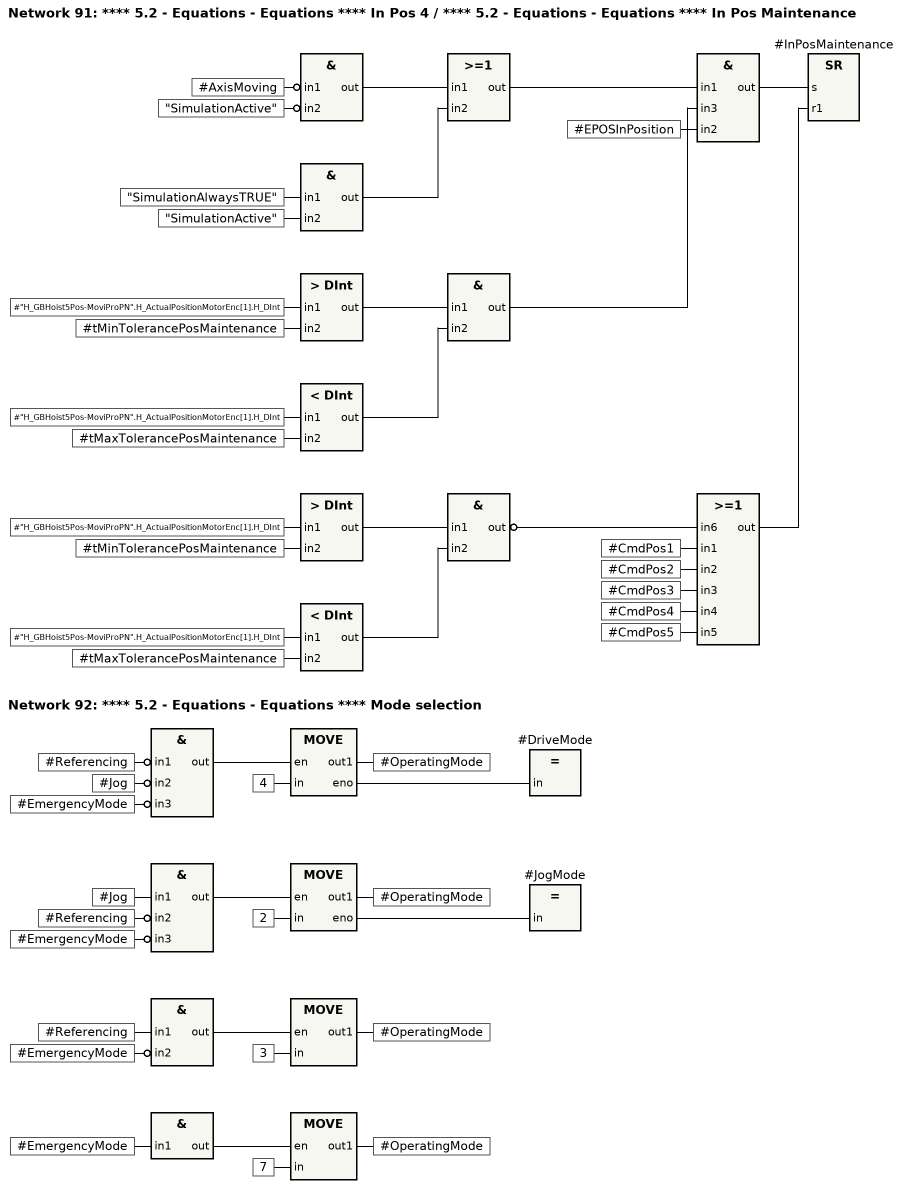
   IF ((NOT #AxisMoving AND NOT "SimulationActive") OR ("SimulationAlwaysTRUE" AND "SimulationActive")) AND (#"H_GBHoist5Pos-MoviProPN".H_ActualPositionMotorEnc[1].H_DInt > #tMinTolerancePosMaintenance) AND (#"H_GBHoist5Pos-MoviProPN".H_ActualPositionMotorEnc[1].H_DInt < #tMaxTolerancePosMaintenance) AND #EPOSInPosition THEN
       #InPosMaintenance := TRUE;   // SR flip-flop
   END_IF;
   IF NOT ((#"H_GBHoist5Pos-MoviProPN".H_ActualPositionMotorEnc[1].H_DInt > #tMinTolerancePosMaintenance) AND (#"H_GBHoist5Pos-MoviProPN".H_ActualPositionMotorEnc[1].H_DInt < #tMaxTolerancePosMaintenance)) OR #CmdPos1 OR #CmdPos2 OR #CmdPos3 OR #CmdPos4 OR #CmdPos5 THEN
       #InPosMaintenance := FALSE;
   END_IF;
END_REGION

REGION Network 92: **** 5.2 - Equations - Equations **** Mode selection
   #_w1 := NOT #Referencing AND NOT #Jog AND NOT #EmergencyMode;
   IF #_w1 THEN #OperatingMode := 4; END_IF;
   #DriveMode := #_w1;
   #_w2 := #Jog AND NOT #Referencing AND NOT #EmergencyMode;
   IF #_w2 THEN
       #OperatingMode := 2;   // Mode selection bits mode: 0=Default 1=Speed control 2=Jog mode 3=Referencing mode 4=Positioning mode 5=Positioning mode - touch probe 6=Speed synchronization 7=Emergency mode _
   END_IF;
   #JogMode := #_w2;
   IF #Referencing AND NOT #EmergencyMode THEN #OperatingMode := 3; END_IF;
   IF #EmergencyMode THEN #OperatingMode := 7; END_IF;
END_REGION

REGION Network 93: **** 5.2 - Equations - Equations **** Start command
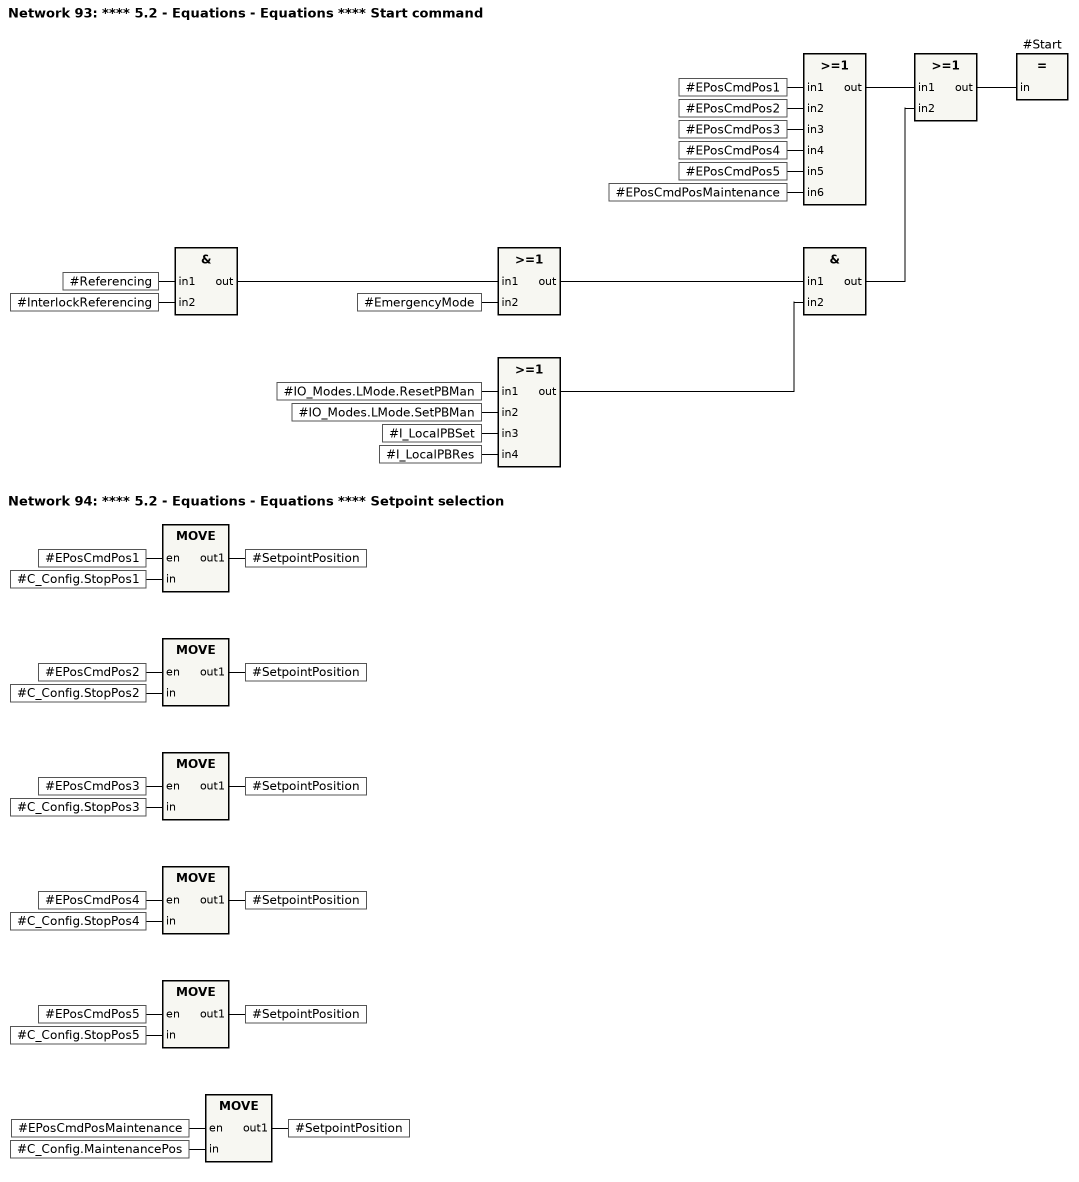
   #Start := #EPosCmdPos1 OR #EPosCmdPos2 OR #EPosCmdPos3 OR #EPosCmdPos4 OR #EPosCmdPos5 OR #EPosCmdPosMaintenance OR (((#Referencing AND #InterlockReferencing) OR #EmergencyMode) AND (#IO_Modes.LMode.ResetPBMan OR #IO_Modes.LMode.SetPBMan OR #I_LocalPBSet OR #I_LocalPBRes));
END_REGION

REGION Network 94: **** 5.2 - Equations - Equations **** Setpoint selection
   IF #EPosCmdPos1 THEN #SetpointPosition := #C_Config.StopPos1; END_IF;
   IF #EPosCmdPos2 THEN #SetpointPosition := #C_Config.StopPos2; END_IF;
   IF #EPosCmdPos3 THEN #SetpointPosition := #C_Config.StopPos3; END_IF;
   IF #EPosCmdPos4 THEN #SetpointPosition := #C_Config.StopPos4; END_IF;
   IF #EPosCmdPos5 THEN #SetpointPosition := #C_Config.StopPos5; END_IF;
   IF #EPosCmdPosMaintenance THEN #SetpointPosition := #C_Config.MaintenancePos; END_IF;
END_REGION

REGION Network 95: **** 7.3 - Submodule - Machine **** Motorloop
   // Motor loop
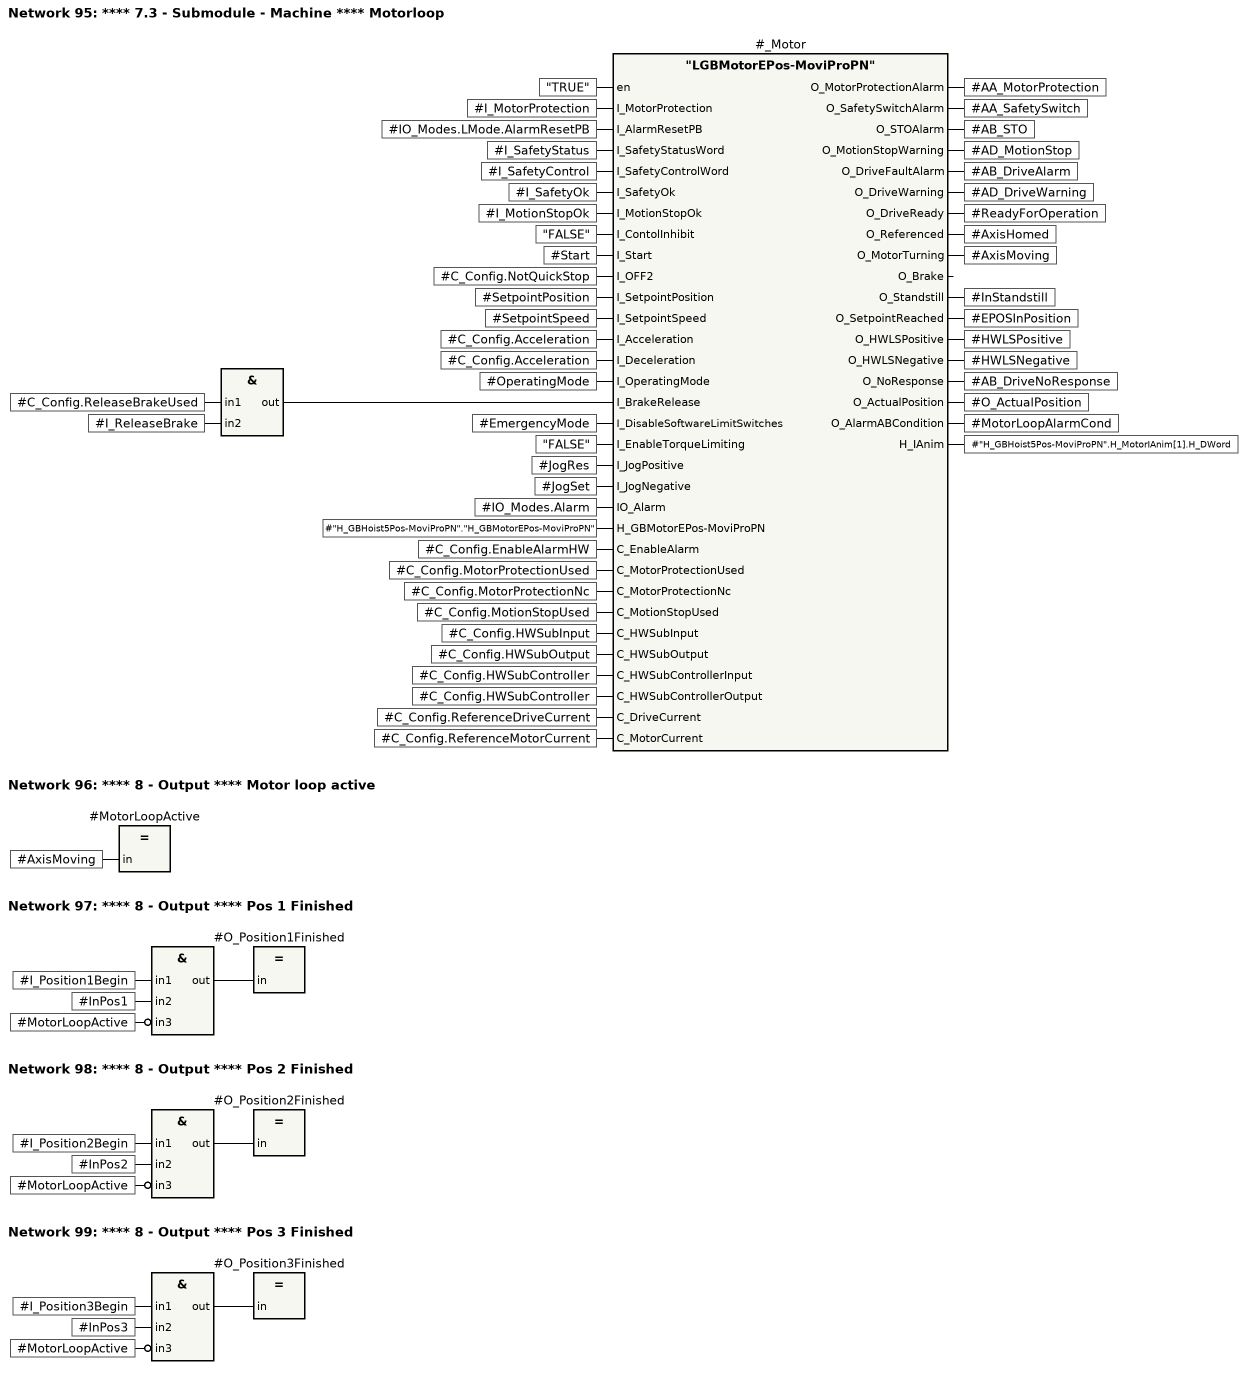
   IF "TRUE" THEN
       #_Motor(I_MotorProtection := #I_MotorProtection,   // "LGBMotorEPos-MoviProPN": Quick stop "I_OFF2" : ^ Speed (%) Stop signal at 5s l / 100% l______________/_ l \ \ l \ \ l \ \ l \ \ 0% l___________________\_____\___________________________> Time (s) l OFF2 OFF1 (regular start stop) 7s 10s ************************************************************************************ "I_SetpointSpeed" , "I_Acceleration", "I_Deceleration": Speed Target speed (user unit) ^ / l ____/____ l / \ l / \ l____/ \____ l--------------------------------------------------> t (s) Speed (user unit) ^ Acceleration l l _________ l l / \ l l/ \ l____/ \____ l--------------------------------------------------> t (s) Speed (user unit) ^ Deceleration l _________ l l / \ l l / \l l____/ \____ l--------------------------------------------------> t (s) ************************************************************************************ Mode selection bits "I_OperatingMode" : mode: 0=Default 1=Speed control 2=Jog mode 3=Referencing mode 4=Positioning mode 5=Positioning mode - touch probe 6=Speed synchronization 7=Emergency mode ************************************************************************************ Software limit switches "I_DisbaleSoftwareLimitSwitches" : The software limit switches are programmed before the hardware limit switches. This will give the drive the possiblility to decelarate accordingly as its knows the distance to these SW LS's from the encoder value. When the referencing is ok it should be impossible to reach the hardware limit switches. Only when there is a faulty referencing then the software limit switches can be behind the hardware limit switch. In that case it is possible to hit the hardware limit switch with full speed. Positive <-- Load --> negative HW LS SW LS _____ SW LS HW LS ____ ____ l_____l ____ ____ l____\ l____\ l_____l /____l /____l OOOOOOOOOOOOOOOOOOOOOOOOOOOOOOOOOOOO ll // \\ ll ll// \\ll ll ll ************************************************************************************ Input "I_EnableTorqueLimiting" : 110% ^ Torque (%) l Torque limited 100% l_______________________________/___________________ torque limit configured in the drive l _ Acceleration l l l l l / l l---- shutdown command l l l/ constant speed l l (error motor blocked) l l l_____/__ l l 0% l___l_________l________________l__l___________________________> Time (s) l l l l l l l / l l l / l_l -100% l __________ /________________________________________ torque limit configured in the drive l Deceleration -110% l ************************************************************************************ Communication handeling is done in the block with the "C_HWSub..." hardware identifiers. SEW Drive ______________ ll __ _ ll__ input telegram ll l__l l_l ll Ol ===============>> PLC ll ll__l ll_____________ll l__l l__l l_ll_l SEW Drive ______________ output telegram ll __ _ ll__ PLC ===============>> ll l__l l_l ll Ol ll ll__l ll_____________ll l__l l__l l_ll_l _
               I_AlarmResetPB := #IO_Modes.LMode.AlarmResetPB,
               I_SafetyStatusWord := #I_SafetyStatus,
               I_SafetyControlWord := #I_SafetyControl,
               I_SafetyOk := #I_SafetyOk,
               I_MotionStopOk := #I_MotionStopOk,
               I_ContolInhibit := "FALSE",
               I_Start := #Start,
               I_OFF2 := #C_Config.NotQuickStop,
               I_SetpointPosition := #SetpointPosition,
               I_SetpointSpeed := #SetpointSpeed,
               I_Acceleration := #C_Config.Acceleration,
               I_Deceleration := #C_Config.Acceleration,
               I_OperatingMode := #OperatingMode,
               I_BrakeRelease := #C_Config.ReleaseBrakeUsed AND #I_ReleaseBrake,
               I_DisableSoftwareLimitSwitches := #EmergencyMode,
               I_EnableTorqueLimiting := "FALSE",
               I_JogPositive := #JogRes,
               I_JogNegative := #JogSet,
               IO_Alarm := #IO_Modes.Alarm,
               "H_GBMotorEPos-MoviProPN" := #"H_GBHoist5Pos-MoviProPN"."H_GBMotorEPos-MoviProPN",
               C_EnableAlarm := #C_Config.EnableAlarmHW,
               C_MotorProtectionUsed := #C_Config.MotorProtectionUsed,
               C_MotorProtectionNc := #C_Config.MotorProtectionNc,
               C_MotionStopUsed := #C_Config.MotionStopUsed,
               C_HWSubInput := #C_Config.HWSubInput,
               C_HWSubOutput := #C_Config.HWSubOutput,
               C_HWSubControllerInput := #C_Config.HWSubController,
               C_HWSubControllerOutput := #C_Config.HWSubController,
               C_DriveCurrent := #C_Config.ReferenceDriveCurrent,
               C_MotorCurrent := #C_Config.ReferenceMotorCurrent,
               O_MotorProtectionAlarm => #AA_MotorProtection,
               O_SafetySwitchAlarm => #AA_SafetySwitch,
               O_STOAlarm => #AB_STO,
               O_MotionStopWarning => #AD_MotionStop,
               O_DriveFaultAlarm => #AB_DriveAlarm,
               O_DriveWarning => #AD_DriveWarning,
               O_DriveReady => #ReadyForOperation,
               O_Referenced => #AxisHomed,
               O_MotorTurning => #AxisMoving,
               O_Standstill => #InStandstill,
               O_SetpointReached => #EPOSInPosition,
               O_HWLSPositive => #HWLSPositive,
               O_HWLSNegative => #HWLSNegative,
               O_NoResponse => #AB_DriveNoResponse,
               O_ActualPosition => #O_ActualPosition,
               O_AlarmABCondition => #MotorLoopAlarmCond,
               H_IAnim => #"H_GBHoist5Pos-MoviProPN".H_MotorIAnim[1].H_DWord);
   END_IF;
END_REGION

REGION Network 96: **** 8 - Output **** Motor loop active
   #MotorLoopActive := #AxisMoving;
END_REGION

REGION Network 97: **** 8 - Output **** Pos 1 Finished
   // Pos 1 Finished
   #O_Position1Finished := #I_Position1Begin AND #InPos1 AND NOT #MotorLoopActive;
END_REGION

REGION Network 98: **** 8 - Output **** Pos 2 Finished
   // Pos 1 Finished
   #O_Position2Finished := #I_Position2Begin AND #InPos2 AND NOT #MotorLoopActive;
END_REGION

REGION Network 99: **** 8 - Output **** Pos 3 Finished
   // Pos 3 Finished
   #O_Position3Finished := #I_Position3Begin AND #InPos3 AND NOT #MotorLoopActive;
END_REGION

REGION Network 100: **** 8 - Output **** Pos 4 Finished
   // Pos 4 Finished
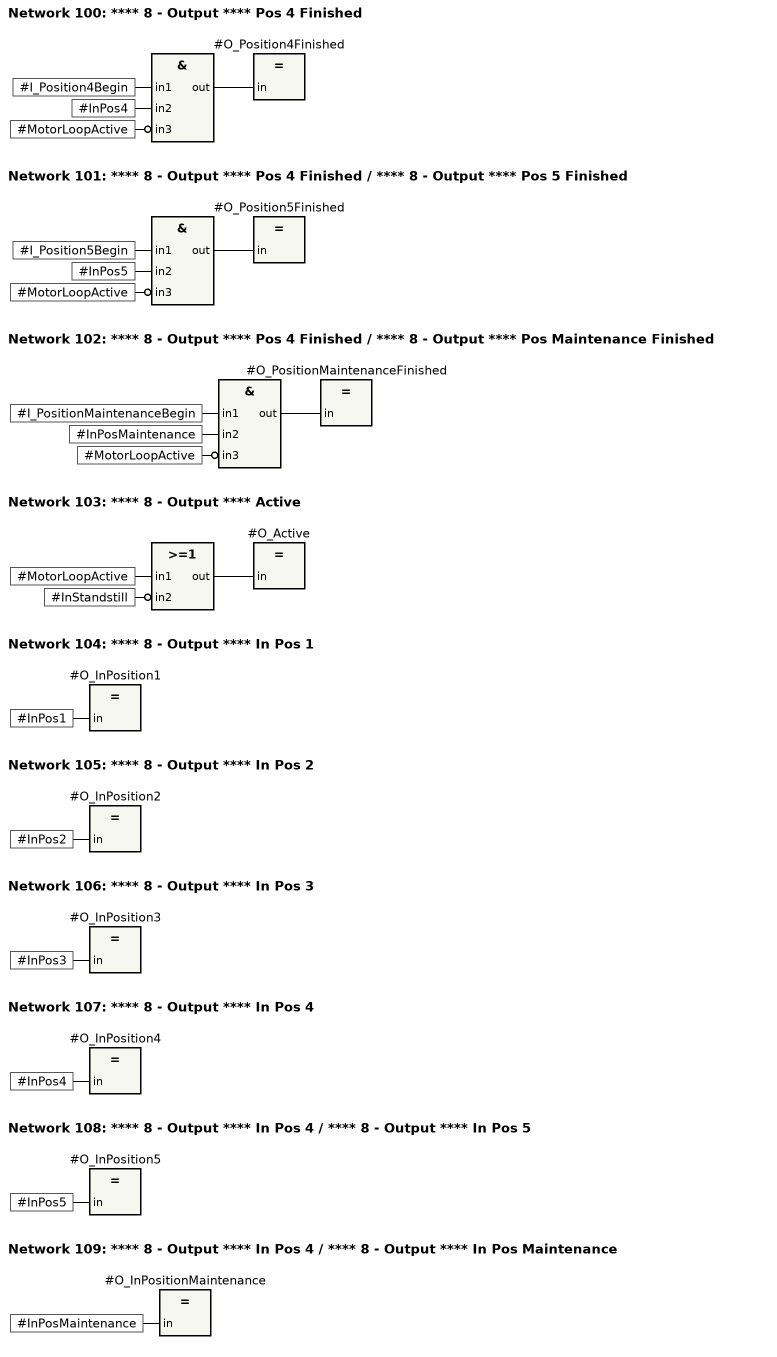
   #O_Position4Finished := #I_Position4Begin AND #InPos4 AND NOT #MotorLoopActive;
END_REGION

REGION Network 101: **** 8 - Output **** Pos 4 Finished / **** 8 - Output **** Pos 5 Finished
   // Pos 4 Finished / Pos 5 Finished
   #O_Position5Finished := #I_Position5Begin AND #InPos5 AND NOT #MotorLoopActive;
END_REGION

REGION Network 102: **** 8 - Output **** Pos 4 Finished / **** 8 - Output **** Pos Maintenance Finished
   // Pos 4 Finished
   #O_PositionMaintenanceFinished := #I_PositionMaintenanceBegin AND #InPosMaintenance AND NOT #MotorLoopActive;
END_REGION

REGION Network 103: **** 8 - Output **** Active
   // Active
   #O_Active := #MotorLoopActive OR NOT #InStandstill;
END_REGION

REGION Network 104: **** 8 - Output **** In Pos 1
   // In Pos 1
   #O_InPosition1 := #InPos1;
END_REGION

REGION Network 105: **** 8 - Output **** In Pos 2
   // In Pos 2
   #O_InPosition2 := #InPos2;
END_REGION

REGION Network 106: **** 8 - Output **** In Pos 3
   // In Pos 3
   #O_InPosition3 := #InPos3;
END_REGION

REGION Network 107: **** 8 - Output **** In Pos 4
   // In Pos 4
   #O_InPosition4 := #InPos4;
END_REGION

REGION Network 108: **** 8 - Output **** In Pos 4 / **** 8 - Output **** In Pos 5
   // In Pos 4 / In Pos 5
   #O_InPosition5 := #InPos5;
END_REGION

REGION Network 109: **** 8 - Output **** In Pos 4 / **** 8 - Output **** In Pos Maintenance
   // In Pos 4
   #O_InPositionMaintenance := #InPosMaintenance;
END_REGION

REGION Network 110: **** 8 - Outputs **** LED - Indication / **** 8 - Outputs **** LED - Indication Position1
   // LED - Indication
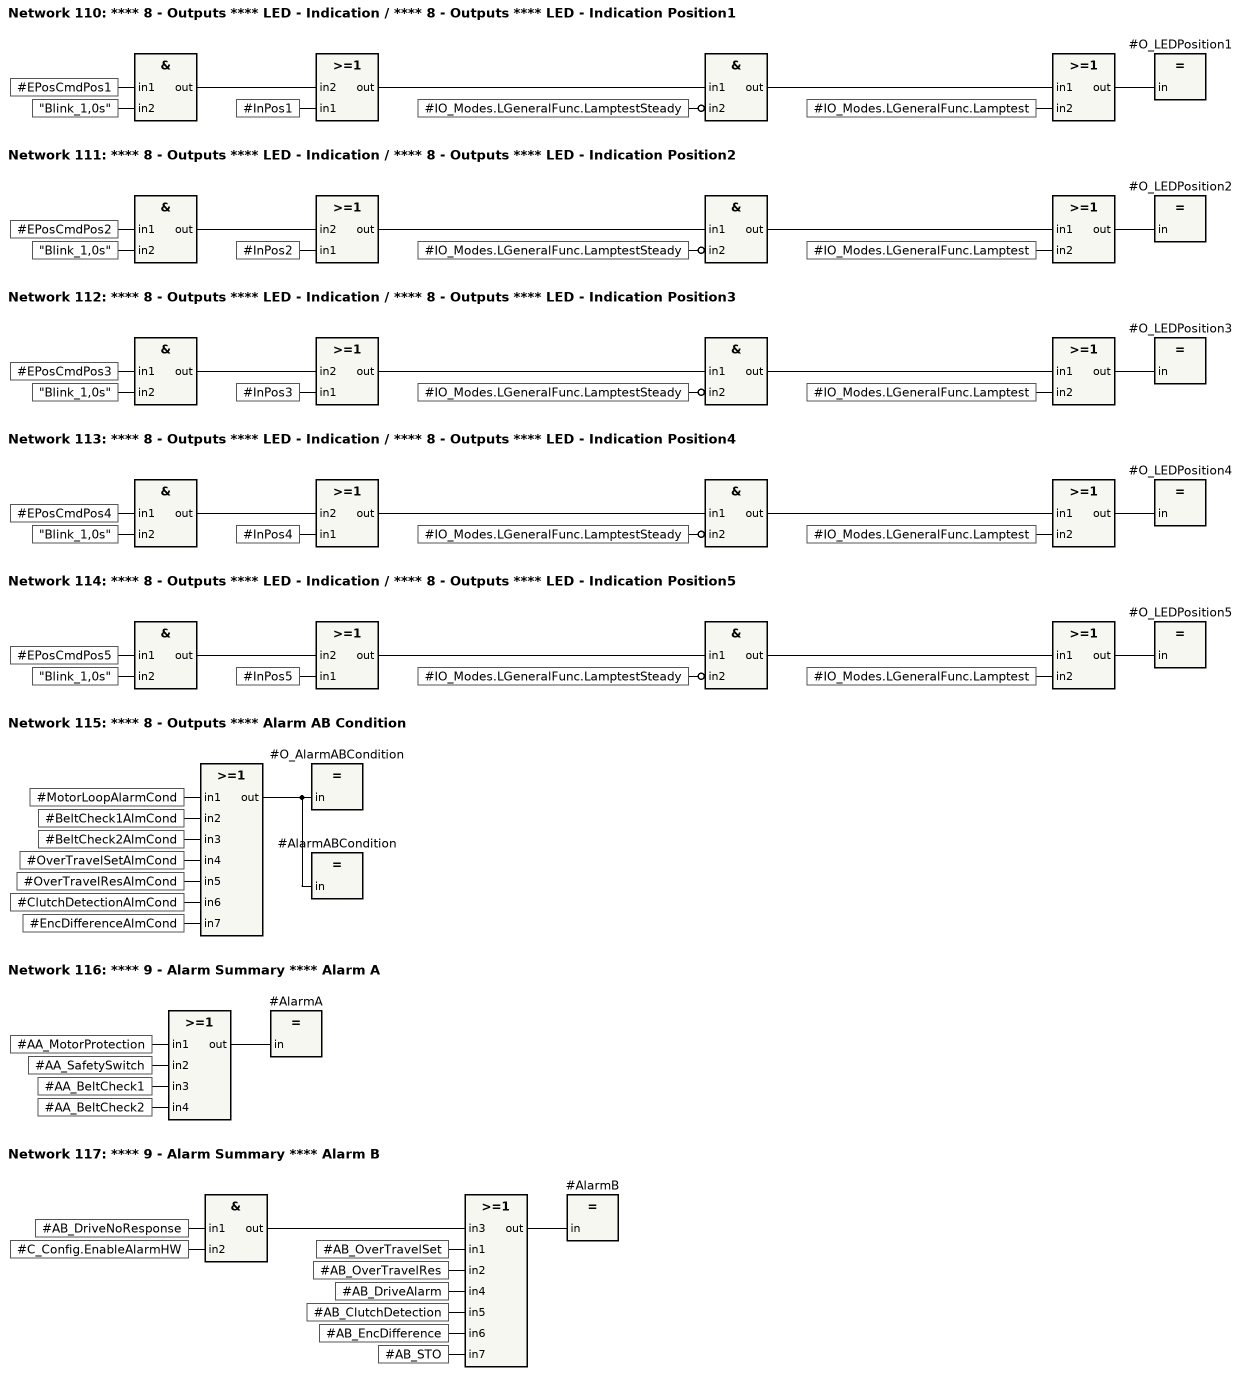
   #O_LEDPosition1 := (((#EPosCmdPos1 AND "Blink_1,0s") OR #InPos1) AND NOT #IO_Modes.LGeneralFunc.LamptestSteady) OR #IO_Modes.LGeneralFunc.Lamptest;
END_REGION

REGION Network 111: **** 8 - Outputs **** LED - Indication / **** 8 - Outputs **** LED - Indication Position2
   // LED - Indication
   #O_LEDPosition2 := (((#EPosCmdPos2 AND "Blink_1,0s") OR #InPos2) AND NOT #IO_Modes.LGeneralFunc.LamptestSteady) OR #IO_Modes.LGeneralFunc.Lamptest;
END_REGION

REGION Network 112: **** 8 - Outputs **** LED - Indication / **** 8 - Outputs **** LED - Indication Position3
   // LED - Indication
   #O_LEDPosition3 := (((#EPosCmdPos3 AND "Blink_1,0s") OR #InPos3) AND NOT #IO_Modes.LGeneralFunc.LamptestSteady) OR #IO_Modes.LGeneralFunc.Lamptest;
END_REGION

REGION Network 113: **** 8 - Outputs **** LED - Indication / **** 8 - Outputs **** LED - Indication Position4
   // LED - Indication
   #O_LEDPosition4 := (((#EPosCmdPos4 AND "Blink_1,0s") OR #InPos4) AND NOT #IO_Modes.LGeneralFunc.LamptestSteady) OR #IO_Modes.LGeneralFunc.Lamptest;
END_REGION

REGION Network 114: **** 8 - Outputs **** LED - Indication / **** 8 - Outputs **** LED - Indication Position5
   // LED - Indication
   #O_LEDPosition5 := (((#EPosCmdPos5 AND "Blink_1,0s") OR #InPos5) AND NOT #IO_Modes.LGeneralFunc.LamptestSteady) OR #IO_Modes.LGeneralFunc.Lamptest;
END_REGION

REGION Network 115: **** 8 - Outputs **** Alarm AB Condition
   // Alarm AB condition
   #O_AlarmABCondition := #MotorLoopAlarmCond OR #BeltCheck1AlmCond OR #BeltCheck2AlmCond OR #OverTravelSetAlmCond OR #OverTravelResAlmCond OR #ClutchDetectionAlmCond OR #EncDifferenceAlmCond;
   #AlarmABCondition := #O_AlarmABCondition;
END_REGION

REGION Network 116: **** 9 - Alarm Summary **** Alarm A
   // Alarm A
   #AlarmA := #AA_MotorProtection OR #AA_SafetySwitch OR #AA_BeltCheck1 OR #AA_BeltCheck2;
END_REGION

REGION Network 117: **** 9 - Alarm Summary **** Alarm B
   // Alarm B
   #AlarmB := (#AB_DriveNoResponse AND #C_Config.EnableAlarmHW) OR #AB_OverTravelSet OR #AB_OverTravelRes OR #AB_DriveAlarm OR #AB_ClutchDetection OR #AB_EncDifference OR #AB_STO;
END_REGION

REGION Network 118: **** 9 - Alarm Summary **** Alarm C
   // Alarm C
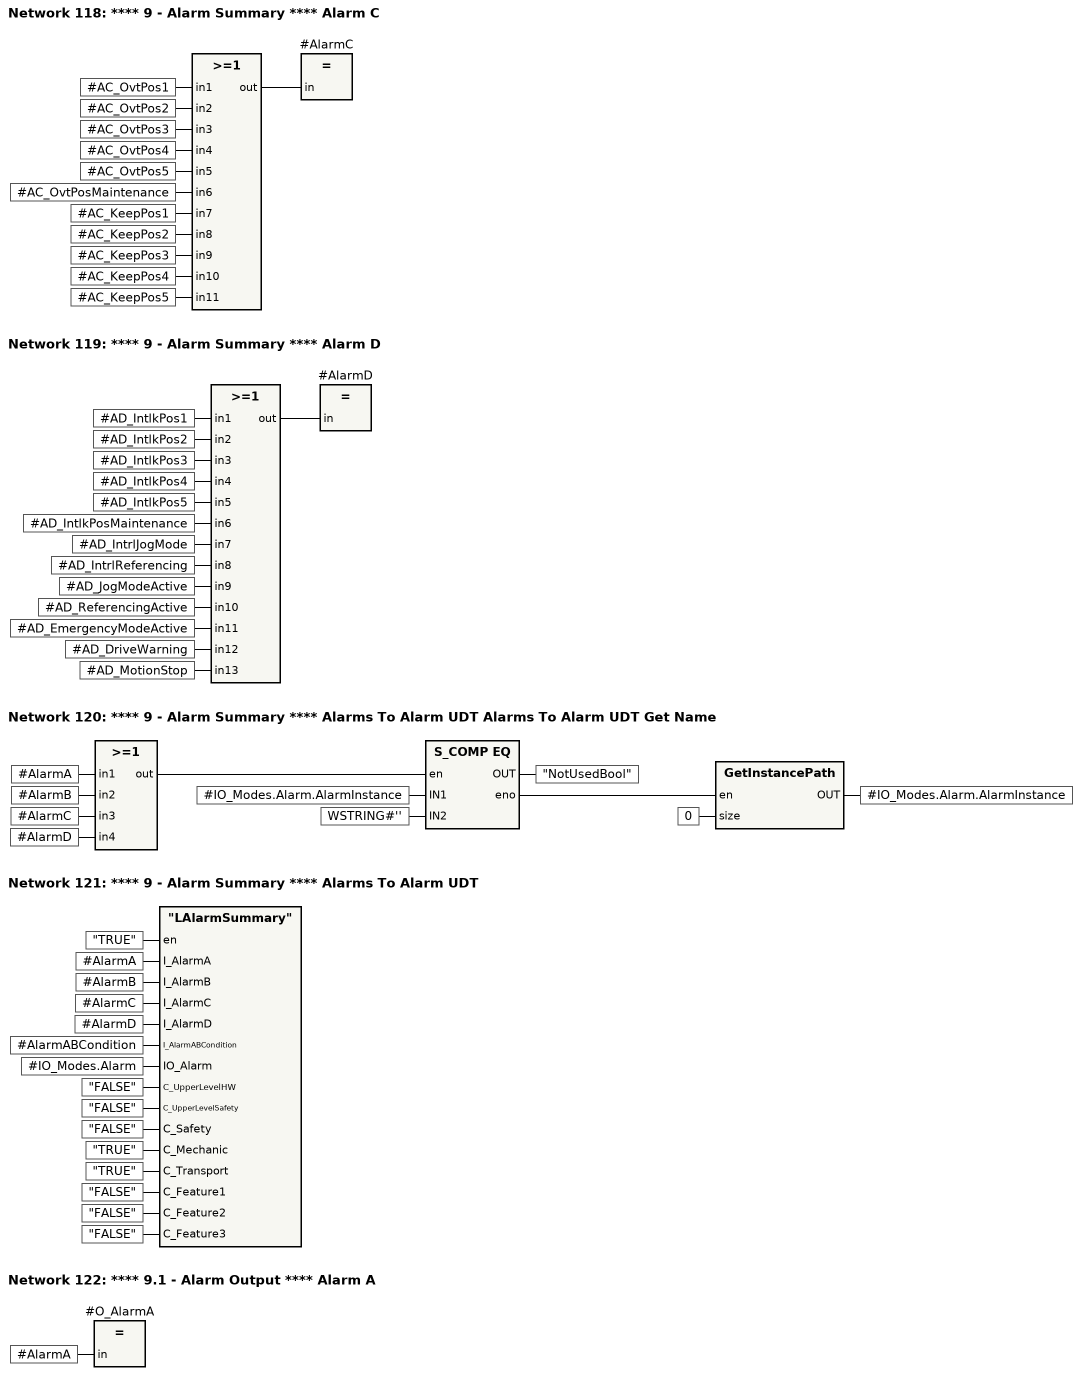
   #AlarmC := #AC_OvtPos1 OR #AC_OvtPos2 OR #AC_OvtPos3 OR #AC_OvtPos4 OR #AC_OvtPos5 OR #AC_OvtPosMaintenance OR #AC_KeepPos1 OR #AC_KeepPos2 OR #AC_KeepPos3 OR #AC_KeepPos4 OR #AC_KeepPos5;
END_REGION

REGION Network 119: **** 9 - Alarm Summary **** Alarm D
   // Alarm D
   #AlarmD := #AD_IntlkPos1 OR #AD_IntlkPos2 OR #AD_IntlkPos3 OR #AD_IntlkPos4 OR #AD_IntlkPos5 OR #AD_IntlkPosMaintenance OR #AD_IntrlJogMode OR #AD_IntrlReferencing OR #AD_JogModeActive OR #AD_ReferencingActive OR #AD_EmergencyModeActive OR #AD_DriveWarning OR #AD_MotionStop;
END_REGION

REGION Network 120: **** 9 - Alarm Summary **** Alarms To Alarm UDT Alarms To Alarm UDT Get Name
   // Alarms To Alarm UDT Alarms To Alarm UDT Get Name
   S_COMP(EN := #AlarmA OR #AlarmB OR #AlarmC OR #AlarmD,
          IN1 := #IO_Modes.Alarm.AlarmInstance,
          IN2 := WSTRING#'',
          OUT => "NotUsedBool",
          ENO => #_w1);
   IF #_w1 THEN GetInstancePath(size := 0, OUT => #IO_Modes.Alarm.AlarmInstance); END_IF;
END_REGION

REGION Network 121: **** 9 - Alarm Summary **** Alarms To Alarm UDT
   // Alarms To Alarm UDT
   IF "TRUE" THEN
       "LAlarmSummary"(I_AlarmA := #AlarmA,
                       I_AlarmB := #AlarmB,
                       I_AlarmC := #AlarmC,
                       I_AlarmD := #AlarmD,
                       I_AlarmABCondition := #AlarmABCondition,
                       IO_Alarm := #IO_Modes.Alarm,
                       C_UpperLevelHW := "FALSE",
                       C_UpperLevelSafety := "FALSE",
                       C_Safety := "FALSE",
                       C_Mechanic := "TRUE",
                       C_Transport := "TRUE",
                       C_Feature1 := "FALSE",
                       C_Feature2 := "FALSE",
                       C_Feature3 := "FALSE");
   END_IF;
END_REGION

REGION Network 122: **** 9.1 - Alarm Output **** Alarm A
   // Alarm A
   #O_AlarmA := #AlarmA;
END_REGION

REGION Network 123: **** 9.1 - Alarm Output **** Alarm B
   // Alarm B
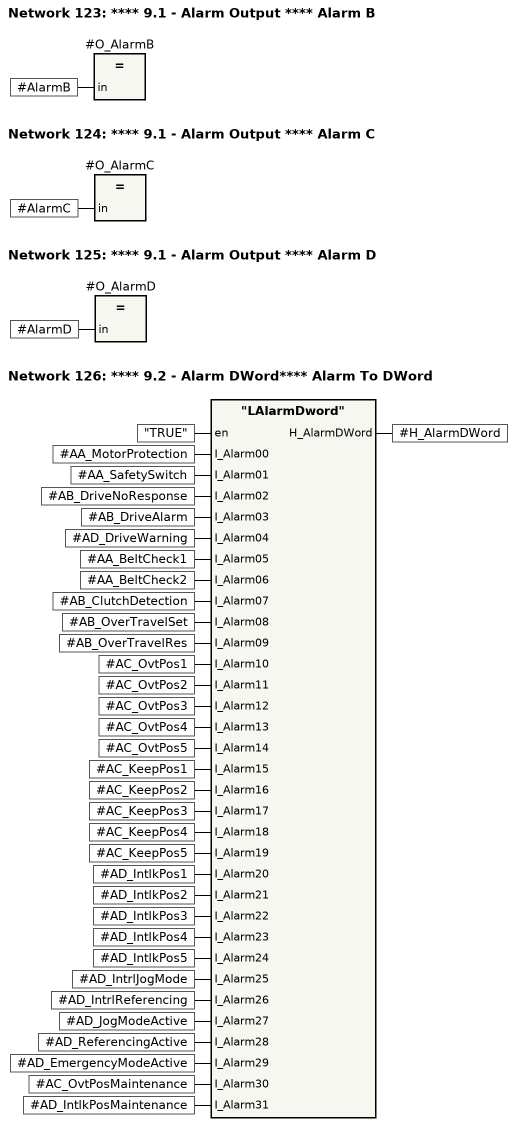
   #O_AlarmB := #AlarmB;
END_REGION

REGION Network 124: **** 9.1 - Alarm Output **** Alarm C
   // Alarm C
   #O_AlarmC := #AlarmC;
END_REGION

REGION Network 125: **** 9.1 - Alarm Output **** Alarm D
   // Alarm D
   #O_AlarmD := #AlarmD;
END_REGION

REGION Network 126: **** 9.2 - Alarm DWord**** Alarm To DWord
   // Alarm To Word
   IF "TRUE" THEN
       "LAlarmDword"(I_Alarm00 := #AA_MotorProtection,
                     I_Alarm01 := #AA_SafetySwitch,
                     I_Alarm02 := #AB_DriveNoResponse,
                     I_Alarm03 := #AB_DriveAlarm,
                     I_Alarm04 := #AD_DriveWarning,
                     I_Alarm05 := #AA_BeltCheck1,
                     I_Alarm06 := #AA_BeltCheck2,
                     I_Alarm07 := #AB_ClutchDetection,
                     I_Alarm08 := #AB_OverTravelSet,
                     I_Alarm09 := #AB_OverTravelRes,
                     I_Alarm10 := #AC_OvtPos1,
                     I_Alarm11 := #AC_OvtPos2,
                     I_Alarm12 := #AC_OvtPos3,
                     I_Alarm13 := #AC_OvtPos4,
                     I_Alarm14 := #AC_OvtPos5,
                     I_Alarm15 := #AC_KeepPos1,
                     I_Alarm16 := #AC_KeepPos2,
                     I_Alarm17 := #AC_KeepPos3,
                     I_Alarm18 := #AC_KeepPos4,
                     I_Alarm19 := #AC_KeepPos5,
                     I_Alarm20 := #AD_IntlkPos1,
                     I_Alarm21 := #AD_IntlkPos2,
                     I_Alarm22 := #AD_IntlkPos3,
                     I_Alarm23 := #AD_IntlkPos4,
                     I_Alarm24 := #AD_IntlkPos5,
                     I_Alarm25 := #AD_IntrlJogMode,
                     I_Alarm26 := #AD_IntrlReferencing,
                     I_Alarm27 := #AD_JogModeActive,
                     I_Alarm28 := #AD_ReferencingActive,
                     I_Alarm29 := #AD_EmergencyModeActive,
                     I_Alarm30 := #AC_OvtPosMaintenance,
                     I_Alarm31 := #AD_IntlkPosMaintenance,
                     H_AlarmDWord => #H_AlarmDWord);
   END_IF;
END_REGION

REGION Network 127: **** 9.2 - Alarm DWord**** Alarm To DWord
   // Alarm To Word
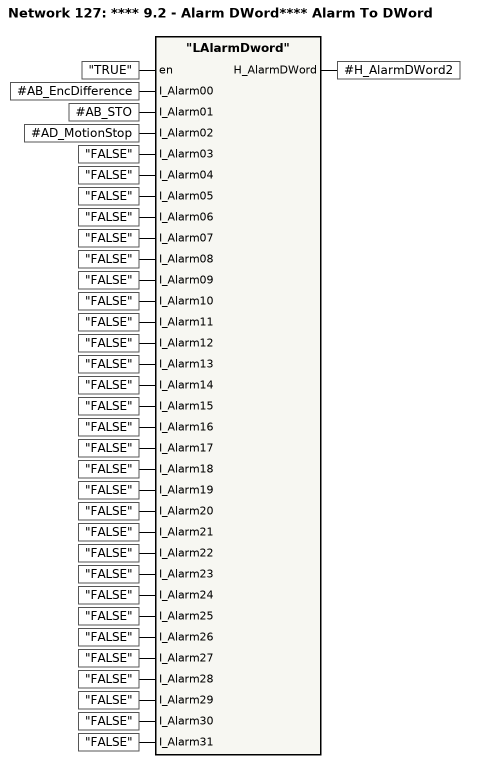
   IF "TRUE" THEN
       "LAlarmDword"(I_Alarm00 := #AB_EncDifference,
                     I_Alarm01 := #AB_STO,
                     I_Alarm02 := #AD_MotionStop,
                     I_Alarm03 := "FALSE",
                     I_Alarm04 := "FALSE",
                     I_Alarm05 := "FALSE",
                     I_Alarm06 := "FALSE",
                     I_Alarm07 := "FALSE",
                     I_Alarm08 := "FALSE",
                     I_Alarm09 := "FALSE",
                     I_Alarm10 := "FALSE",
                     I_Alarm11 := "FALSE",
                     I_Alarm12 := "FALSE",
                     I_Alarm13 := "FALSE",
                     I_Alarm14 := "FALSE",
                     I_Alarm15 := "FALSE",
                     I_Alarm16 := "FALSE",
                     I_Alarm17 := "FALSE",
                     I_Alarm18 := "FALSE",
                     I_Alarm19 := "FALSE",
                     I_Alarm20 := "FALSE",
                     I_Alarm21 := "FALSE",
                     I_Alarm22 := "FALSE",
                     I_Alarm23 := "FALSE",
                     I_Alarm24 := "FALSE",
                     I_Alarm25 := "FALSE",
                     I_Alarm26 := "FALSE",
                     I_Alarm27 := "FALSE",
                     I_Alarm28 := "FALSE",
                     I_Alarm29 := "FALSE",
                     I_Alarm30 := "FALSE",
                     I_Alarm31 := "FALSE",
                     H_AlarmDWord => #H_AlarmDWord2);
   END_IF;
END_REGION
END_FUNCTION_BLOCK
